# B&R Automation Studio project TD52 (part 22)

### module_AG.typ
```iecst
TYPE
	IN_AG_struct : 	STRUCT
		bCust_Dem_FreshOilPump : BOOL; (*Customized demand for fresh oil pump*) (*OldName:new V4.14; Cycle:5*)
		bCust_Dem_WasteOilPump : BOOL; (*Customized demand for waste oil pump*) (*OldName:new V4.14; Cycle:5*)
		bCust_Dem_OilFillValve : BOOL; (*Customized demand for oil fill valve*) (*OldName:new V4.14; Cycle:5*)
		bMsg1061 : BOOL; (* *) (*OldName:; Cycle:;*)
		tL_FreshOilTank : HALioAi_Type; (*Tank Level measurement input*) (*OldName: NewPv V4.12*)
		tL_WasteOilTank : HALioAi_Type; (*Tank Level measurement input*) (*OldName: NewPv V4.12*)
		tL_DayOilTank : HALioAi_Type; (*Tank Level measurement input*) (*OldName: NewPv V4.12*)
		tCDP_Op : HALioDi_Type; (*Di condensor pump failure*) (*OldName:GCB_ON; Cycle:5*)
		tFOP_Op : HALioDi_Type; (*DI fresh oil pump operating*) (*OldName:GCB_ON; Cycle:5*)
		tL_DayOilSump_Hi : HALioDi_Type; (*DI day oil tank oil collector pan high*) (*OldName:GCB_ON; Cycle:5*)
		tDayOilTank_Leck : HALioDi_Type; (*DI leckage day oil tank*) (*OldName:GCB_ON; Cycle:5*)
		tL_DayOilTank_Hi : HALioDi_Type; (*DI day oil tank high*) (*OldName:GCB_ON; Cycle:5*)
		tAuxV_Aux_ok : HALioDi_Type; (*DI voltage ok auxiliaries panel*) (*OldName:GCB_ON; Cycle:5*)
		tAuxV_ModIf_ok : HALioDi_Type; (*DI release auxiliaries module interface*) (*OldName:GCB_ON; Cycle:5*)
		tAB2AG : AmmBase2MM; (*AmmBase2MM*) (*OldName:new; Cycle:5*)
		tPB2MM : ParaBase2MM_type; (*ParaBase2MM*) (*OldName:new; Cycle:5*)
		iIdx_OMSS : INT; (*engine operation mode selection*) (*OldName:new; Cycle:5*)
		bIgn_Run : BOOL; (*ignition operating*) (*OldName:ZIB; Cycle:5*)
		bDemScavVa : BOOL; (* demand scavenging valve *) (*OldName:ANF_SPKL; Cycle:5*)
		b_ST_DemIgn : BOOL; (* Demand starter from ignition *) (*OldName:STARTER_IgnST; Cycle:5*)
		bBlocDelay_ManStart : BOOL; (* delay time next manual start *) (*OldName:T26; Cycle:5*)
		bECW_PreH_Dem_Customized : BOOL; (* engine cooling water preheating demand customized *) (*OldName:new; Cycle:5*)
		bEng_Aux_Dem_TOF : BOOL; (* demand auxiliaries with cool down time *) (*OldName:T12; Cycle:5*)
		bEG_BoVaOpened : BOOL; (* exhaust gas boiler valve opened *) (*OldName:M_KKAUF; Cycle:5*)
		bEG_ByVaOpened : BOOL; (* exhaust gas bypass valve opened *) (*OldName:M_BKAUF; Cycle:5*)
		bEO_PrelubeDemIgn : BOOL; (* demand Prelubricating from ignition *) (*OldName:PRELUBE_IgnST; Cycle:5*)
		tGCB_On : HALioDi_Type; (*DI generator circuit breaker closed*) (*OldName:GCB_ON; Cycle:5*)
		bGT_Rel : BOOL; (* Release gas train *) (*OldName:FG_GST; Cycle:5*)
		bGT_TypSwhActive : BOOL; (* Gas type switching active *) (*OldName:GASUM; Cycle:5*)
		bGT1_Check : BOOL; (* Gas train check 1 *) (*OldName:T88; Cycle:5*)
		bGT1_CheckOK : BOOL; (* Gas train 1 check OK *) (*OldName:M_GAS1OK; Cycle:5*)
		bGT2_Check : BOOL; (* Gas train check 2 *) (*OldName:T90; Cycle:5*)
		bGT2_CheckOK : BOOL; (* Gas train 2 check OK *) (*OldName:M_GAS2OK; Cycle:5*)
		bEng_Aux_Dem : BOOL; (*engine auxiliaries demand*) (*OldName:M_ANFHBT; Cycle:5*)
		bEng_Aux_Dem_CDR : BOOL; (*engine auxiliaries demand with cool down run*) (*OldName:ANFHBT; Cycle:5*)
		bEng_Dem : BOOL; (* module demanded *) (*OldName:M_AGFD; Cycle:5*)
		bEng_Dem_Aut_SUpF : BOOL; (* engine demand automatic startup failure *) (*OldName:BRI; Cycle:5*)
		bEng_Dem_Man_SUpF : BOOL; (* engine demand manual startup failure *) (*OldName:BRI_H; Cycle:5*)
		bEng_Dem_EPS : BOOL; (* engine demand for emergency operation *) (*OldName:M_NANF; Cycle:5*)
		bEng_Dem_Man : BOOL; (* engine demand manual *) (*OldName:M_ANF_H; Cycle:5*)
		bEng_MonOff : BOOL; (* engine monitoring OFF at startup *) (*OldName:T9; Cycle:5*)
		bEng_Rel : BOOL; (* engine release *) (*OldName:M_FG_MOT; Cycle:5*)
		bEng_RPSDem : BOOL; (* engine demanded  *) (*OldName:A_AGFD; Cycle:5*)
		tEng_Run : HALioDo_Type; (* engine operating state *) (*OldName:BTRB; Cycle:5*)
		bEng_SU_Man : BOOL; (* engine startup manual *) (*OldName:M_HSTART; Cycle:5*)
		bEng_SU_Aut : BOOL; (* engine startup automatic *) (*OldName:M7_6; Cycle:5*)
		bGV_On : BOOL; (* command open gas valves *) (*OldName:M_GASV; Cycle:5*)
		bMainsReturn : BOOL; (* mains return *) (*OldName:NWK; Cycle:5*)
		tMCB_On : HALioDi_Type; (*DI mains circuit breaker closed*) (*OldName:MCB_ON; Cycle:5*)
		bMsg1019 : BOOL; (* pressure engine cooling water low *) (*OldName:M_KDMI; Cycle:5*)
		bMsg1027 : BOOL; (* failure gas train 1 *) (*OldName:M_GST1; Cycle:5*)
		bMsg1029 : BOOL; (* failure gas train 2 *) (*OldName:M_GST2; Cycle:5*)
		bMsg1031 : BOOL; (* safety loop *) (*OldName:M_SIS; Cycle:5*)
		bN2_ScavCoPrelubeOn : BOOL; (* N2 scavenging command prelubrication ON *) (*OldName:PRELUBE_SC; Cycle:5*)
		bN2_ScavCoStarterOn : BOOL; (* N2 scavening command starter ON *) (*OldName:STARTER_SC; Cycle:5*)
		bOnly_Island : BOOL; (* only island operation *) (*OldName:REIN_INSEL; Cycle:5*)
		bOtherGenParallel : BOOL; (* other generator parallel *) (*OldName:other_gen_parallel; Cycle:5*)
		bP_Red_Active : BOOL; (* power reduction active - any kind *) (*OldName:PredAkt; Cycle:5*)
		bRel_ScavN2 : BOOL; (* conditions for scavenge with N2 *) (*OldName:FG_N2; Cycle:5*)
		bRelEngOp_OilSkid : BOOL; (*release engine operation from Oil Skid*) (*OldName:rel_EngOp_LOS; Cycle:5*)
		bRelEngTurn_OilSkid : BOOL; (*release engine barring gear (Durchdrehvorrichtung) from Oil Skid*) (*OldName:tPr_GenJOS_Ok; Cycle:5*)
		bScavFinished : BOOL; (* scavenging cycle finished  *) (*OldName:SPUEL_AB; Cycle:5*)
		tScavVaClosed : HALioDi_Type; (*DI scavenging valve closed*) (*OldName:SPK_ZU; Cycle:5*)
		rN_EngAct : REAL; (* engine speed actual [1/min] *) (*OldName:n_ist; Cycle:5*)
		rP_Act_Norm_Filt : REAL; (* actual power related to rP_Nom filtered T=1s *) (*OldName:P_IST; Cycle:5*)
		tAuxV_Eng_ok : HALioDi_Type; (* DI auxiliary voltage engine ok *) (*OldName:DI_AuxV_Eng_ok; Cycle:5*)
		tCCWP_Op : HALioDi_Type; (* DI charge cooling water pump operating (P.07-M-003) *) (*OldName:RM_GKP; Cycle:5*)
		tECWPrehV_Opened : HALioDi_Type; (* DI engine cooling water preheating valve opened *) (*OldName:new; Cycle:5*)
		tECWP_FC_Rdy : HALioDi_Type; (* DI engine cooling water pump frequency converter ready for operation *) (*OldName:MKP_FU_rdy; Cycle:5*)
		tECWP_Op : HALioDi_Type; (* DI engine cooling water pump operating *) (*OldName:RM_MKWP; Cycle:5*)
		tEngTurn : HALioDi_Type; (* DI engine turn equipment active *) (*OldName:DI_TURN1; Cycle:5*)
		tEngTurn2 : HALioDi_Type; (* DI engine turn equipment active *) (*OldName:DI_TURN2; Cycle:5*)
		tEO_Level_Hi : HALioDi_Type; (* DI engine oil level high from level switch  *) (*OldName:OMAX; Cycle:5*)
		tEO_Level_Lo : HALioDi_Type; (* DI engine oil level low from level switch  *) (*OldName:OMIN; Cycle:5*)
		tEO_Level_Lo_TC2 : HALioDi_Type; (* DI engine oil level low from level switch  *) (*OldName:OMIN; Cycle:2*)
		tEO_Refill : HALioDi_Type; (* DI engine oil refill ON from level switch *) (*OldName:OELV; Cycle:5*)
		tEOP_DemExt : HALioDi_Type; (* DI engine oil pump demand from external *) (*OldName:ANF_NKOP; Cycle:5*)
		tEOP_Op : HALioDi_Type; (* DI engine oil pump operating *) (*OldName:RM_VSP; Cycle:5*)
		tEOP1AC_CB_trip : HALioDi_Type; (* DI engine oil pump 1 AC circuit breaker trip *) (*OldName:DI_EOP1AC_CB_trip; Cycle:5*)
		tFireAlarm : HALioDi_Type; (* DI fire alarm *) (*OldName:BAL; Cycle:5*)
		tFS_ECW : HALioDi_Type; (* DI flow switch engine cooling water *) (*OldName:DI_FS_ECW; Cycle:5*)
		tGasAlarm : HALioDi_Type; (* DI gas alarm *) (*OldName:GAL; Cycle:5*)
		tGasPreAlarm : HALioDi_Type; (* DI gas pre alarm *) (*OldName:GALV; Cycle:5*)
		tGF_OilSystem : HALioDi_Type; (*DI general failure oil system*) (*OldName:newPV; Cycle:5*) (*STM 2*)
		tGT1_SafeDevOK : HALioDi_Type; (* DI Gassafety device 1 *) (*OldName:F_GAS1; Cycle:5*)
		tGT2_SafeDevOK : HALioDi_Type; (* DI Gassafety device 2 *) (*OldName:F_GAS2; Cycle:5*)
		tHWP_Op : HALioDi_Type; (* DI heating water pump operating (P.06-M-001) *) (*OldName:RM_HWP; Cycle:5*)
		tL_FreshOilTank_Hi : HALioDi_Type; (*DI fresh oil tank level high*) (*OldName:newPV; Cycle:5*) (*STM 2*)
		tLeak_FreshOilPump : HALioDi_Type; (*DI leakage fresh oil pump*) (*OldName:newPV; Cycle:5*) (*STM 2*)
		tLeak_FreshOilTank : HALioDi_Type; (*DI leakage fresh oil tank*) (*OldName:newPV; Cycle:5*) (*STM 2*)
		tLeak_WasteOilPump : HALioDi_Type; (*DI leakage waste oil pump*) (*OldName:newPV; Cycle:5*) (*STM 2*)
		tLeak_WasteOilTank : HALioDi_Type; (*DI leakage waste oil tank*) (*OldName:newPV; Cycle:5*) (*STM 2*)
		tMainsStartDevFail : HALioDi_Type; (* DI mains start device failure *) (*OldName:ST_NST; Cycle:5*)
		tMainsStartDevOk : HALioDi_Type; (* DI mains starting device OK *) (*OldName:FG_NST; Cycle:5*)
		tN2_GV1_Closed : HALioDi_Type; (* DI N2 gas valve 1 closed status *) (*OldName:N2V1_ZU; Cycle:5*)
		tN2_GV2_Closed : HALioDi_Type; (* DI N2 gas valve 2 closed status *) (*OldName:N2V2_ZU; Cycle:5*)
		tInAirER_Lou1Opened : HALioDi_Type; (* DI intake air engine room louver 1 opened*) (*OldName:ZJAL1_O; Cycle:5*)
		tInAirER_Lou2Opened : HALioDi_Type; (* DI intake air engine room louver 2 opened*) (*OldName:ZJAL2_O; Cycle:5*)
		tOF_FreshOilTank : HALioDi_Type; (*DI overfill prevention device fresh oil tank*) (*OldName:newPV; Cycle:5*) (*STM 2*)
		tOF_WasteOilTank : HALioDi_Type; (*DI overfill prevention device waste oil tank*) (*OldName:newPV; Cycle:5*) (*STM 2*)
		tOutAirER_LouOpened : HALioDi_Type; (* DI outlet air engine room louver opened*) (*OldName:AJAL_O; Cycle:5*)
		tP_Heat_Imp : HALioDi_Type; (*heating power engine heat water circuit impulse*) (*STM 2*)
		tPr_CC : HALioAi_Type; (* AI pressure crank case [bar] *) (*OldName:AI_KGD; Cycle:5*)
		tPr_EngLubOil : HALioAi_Type; (*AI: Oil pressure engine lube oil - last lubr. point [bar] M.03-PI-001*) (*OldName:ODR_WE; Cycle:5*)
		tRelAux : HALioDi_Type; (* DI release engine operation from auxiliaries with monitoring *) (*OldName:FG_HBT; Cycle:5*)
		tRelAuxNoMon : HALioDi_Type; (* DI release engine operation from auxiliaries without bridging for blackout start *) (*OldName:FG_HBT2; Cycle:5*)
		tRelMainGVext : HALioDi_Type; (* DI release main gas valve from external *) (*OldName:FG_HGV_ext; Cycle:5*)
		tT_ECW : HALioAi_Type; (* AI temperature engine cooling water [°C] M.04-TI-001 *) (*OldName:ANA.KWT; Cycle:5*)
		tT_ECW_Mod_In : HALioAi_Type; (*temperature engine cooling water, engine cooling water module inlet M.04-TI-003*) (*OldName:newPv; Cycle:5;*)
		tT_ECW_PreH_Hi : HALioDi_Type; (* TS: temperature engine cooling water preheating high M.04-TI-081*) (*OldName:mkw_preh_warn; Cycle:5*)
		tT_ECW_PreH_HiHi : HALioDi_Type; (* TS: temperature engine cooling water preheating high high M.04-TI-026*) (*OldName:mkw_preh_alarm; Cycle:5*)
		tTCOP_Op : HALioDi_Type; (* DI turbo charger oil pump operating *) (*OldName:RM_TLP; Cycle:5*)
		tU_StarterBat_Lo : HALioDi_Type; (* DI voltage starter battery low *) (*OldName:STBM; Cycle:5*)
		tU_Starter_engage1 : HALioAi_Type; (*Start motor 1 function voltage*)
		tU_Starter_engage2 : HALioAi_Type; (*Start motor 2 function voltage*)
		tU_Starter_engage3 : HALioAi_Type; (*Start motor 3 function voltage*)
		tAuxFail : HALioDi_Type; (*DI auxilaries failure*) (*OldName:ST_HBT; Cycle:5*)
		tECW_PreHV_Closed : HALioDi_Type; (*DI engine cooling water preheating valve status closed M.04-YCS-002*) (*OldName:DI_ECWV_Closed; Cycle:5*)
		tECW_PreHV_Opened : HALioDi_Type; (*DI engine cooling water preheating valve status opened M.04-YCS-002*) (*OldName:DI_ECWV_Open; Cycle:5*)
		tL_ECW_Lo : HALioDi_Type; (*DI engine cooling water level low*) (*OldName:KSMI_W; Cycle:5*)
		tL_ECW_LoLo : HALioDi_Type; (*DI engine cooling water level low low*) (*OldName:KSMI; Cycle:5*)
		tEngStartFailure : HALioDi_Type; (*DI engine start failure*) (*OldName:ANLST; Cycle:5*)
		tTransformerWarning : HALioDi_Type; (*DI transformer failure*) (*OldName:ST_TR_W; Cycle:5*)
		tTransformerTrip : HALioDi_Type; (*DI transformer failure*) (*OldName:ST_TR; Cycle:5*)
		tCP_CBTrip : HALioDi_Type; (*DI module and/or interface control panel - circuit breaker tripped*) (*OldName:SIFA_IA; Cycle:5*)
		tIFCP_CBTrip : HALioDi_Type; (*DI interface control panel - circuit breaker tripped*) (*OldName:SIFA_I; Cycle:5*)
		tMCP_CBTrip : HALioDi_Type; (*DI module control panel - circuit breaker tripped*) (*OldName:SIFA_A; Cycle:5*)
		tSafetyLoop_Gas : HALioDi_Type; (*DI safety loop gas ok*) (*OldName:DI_Gas_SL; Cycle:5*)
		tGV1_Open : HALioDo_Type; (*DO open gas valve 1*) (*OldName:GASV1; Cycle:5*)
		tGV2_Open : HALioDo_Type; (*SAFETY PLC: DO open gas valve 2*) (*OldName:GASV2; Cycle:5*) (*V04.14.00.00*)
		tGV3_Open : HALioDo_Type; (*SAFETY PLC: DO open gas valve 3*) (*OldName: new PV; Cycle: 5;*) (*V04.25.00.00*)
		tGV4_Open : HALioDo_Type; (*SAFETY PLC: DO open gas valve 4*) (*OldName: new PV; Cycle: 5;*) (*V04.25.00.00*)
		tDCGA_GV_Open : HALioDo_Type; (*SAFETY PLC: DO open gas valve for decentral gas addition*) (*OldName: new PV; Cycle: 5;*) (*V04.25.00.00*)
		tL_FreshOilTank_Lo : HALioDi_Type; (*DI fresh oil tank level low*) (*OldName:FOTMI; Cycle:5*)
		tL_WasteOilTank_Hi : HALioDi_Type; (*DI waste oil tank level high*) (*OldName:AOTMA; Cycle:5*)
		tAuxOverVoltProt_Ok : HALioDi_Type; (*failure over voltage protection auxiliaries power supply*) (*OldName:DI_AOVP; Cycle:5*)
		tUPS_Ok : HALioDi_Type; (*uninterrupted power supply ok/alarm*) (*OldName:DI_USV_OK; Cycle:5*)
		tSafetyLoop_Eng : HALioDi_Type; (*safety loop engine ok*) (*OldName:RUHE; Cycle:5*)
		tSafetyLoop_EmStop : HALioDi_Type; (*safety loop emergency stop ok*) (*OldName:DI_SIS; Cycle:5*)
		tSafetyLoop_HWC : HALioDi_Type; (*safety loop heat water circuit ok*) (*OldName:RM_HK; Cycle:5*)
		tPr_HW_Lo : HALioDi_Type; (*DI heat water pressure low*) (*OldName:HWD; Cycle:5*)
		tPr_HW_Hi1 : HALioDi_Type; (*DI heat water pressure high*) (*OldName:HWDX1; Cycle:5*)
		tPr_HW_Hi : HALioDi_Type; (*DI heat water pressure high*) (*OldName:HWDX; Cycle:5*)
		tT_HW_Hi1 : HALioDi_Type; (*DI heat water temperature high*) (*OldName:HWTP1; Cycle:5*)
		tT_HW_Hi : HALioDi_Type; (*DI heat water temperature high*) (*OldName:HWTP; Cycle:5*)
		tT_AirIFCP_Hi : HALioDi_Type; (*DI air temperature interface control panel high*) (*OldName:MCP_TEMP; Cycle:5*)
		tPr_TC_EOF_After : HALioAi_Type; (*AI oil pressure after turbocharger oil filter, J920: NUP62/M.03-PI-062 // J6: M.03-PI-063*) (*OldName:OilPress_a_ATL_f; Cycle:5*)
		tEOF_DiffMax : HALioDi_Type; (*DI: Oil filter differential pressure maximum E.03-PDS-001*) (*OldName:ODFM; Cycle:5*)
		tPr_TCOF_EOF_DiffMax : HALioDi_Type; (*DI: Turbo charger oil filter differential pressure maximum M.03-PDS-001*) (*OldName:DI_dp_TCOF_hi; Cycle:5*)
		tPr_EO_Gear_Min : HALioDi_Type; (*DI: Oil pressure low transmission*) (*OldName:GO_DMI; Cycle:5*)
		tT_EO_Gear_Max : HALioDi_Type; (*DI: Oil temperature high transmission*) (*OldName:GO_TMA; Cycle:5*)
		tEO_Supply_Fail : HALioDi_Type; (*DI: Oil supply failure*) (*OldName:ST_OELV; Cycle:5*)
		tPr_EOF_DiffMon : HALioAi_Type; (*AI: Oil pressure before oil filter [bar] M.03-PI-002 (NUP29)*) (*OldName:ssOilPbFilter; OilPress_f_f; Cycle:5*)
		tPr_EOF_After : HALioAi_Type; (*AI: Oil pressure after oil filter [bar] M.03-PI-057 (NUP57)*) (*OldName:OilPress_a_f; Cycle:5*)
		tEO_Quality : HALioAi_Type; (*AI: Oil quality sensor, QTOil1/ AI_ *) (*OldName:OilQual; Cycle:5*)
		tPr_TC_EOF_Before : HALioAi_Type; (*AI: Oil pressure in front of turbocharger oil filter, NUP61/M.03-PI-061*) (*OldName:OilPress_f_ATL_f; Cycle:5*)
		tEO_Level : HALioAi_Type; (*AI: Oil fill level, LS5/M.03-LI-001*) (*OldName:Oil_Fill; Cycle:5*)
		tT_EO : HALioAi_Type; (*AI: Oil temperature M.03-TI-001*) (*OldName:ANA.OTP; Cycle:5*)
		tT_EO_Mod_Out : HALioAi_Type; (*temperature engine oil, oil module outlet M.03-TI-003*) (*OldName:newPv; Cycle:5;*)
		tCnt_Oil_NC150 : HALioAi_Type; (*AI oil counter*) (*OldName:AIOilCounter; Cycle:2*)
		tCnt_Oil_DC2395 : HALioAi_INT_Type; (*AI oil counter circular buffer*) (*OldName:AIOilCounterCircle; Cycle:2*)
		iCnt_OpHours : DINT; (*Operating hours *) (*OldName:betrieb_h; Cycle:5*)
		rP_Nom : REAL; (*Nominal electric power [kW], depends on gastype*) (*OldName:p_nenn; Cycle:5*)
		tT_EO_Preheating : HALioAi_Type; (*engine oil temperature preheating, NUT78/M.03-TI-078*) (*OldName:OilTemp_preh; Cycle:5*)
		tT_EO_Pan : HALioAi_Type; (*engine oil temperature oil pan, M.03-TI-002*) (*OldName:AI_t_OilPan; Cycle:5*)
		tT_EO_PreH_Hi : HALioDi_Type; (*engine oil preheating max.warning(temp.limiter) M.03-TS-072*) (*OldName:DI_EO_PreH_w; Cycle:5*)
		tT_EO_PreH_HiHi : HALioDi_Type; (*engine oil preheating max.alarm(temp.limiter) M.03-TS-080*) (*OldName:DI_EO_PreH_a; Cycle:5*)
		tT_EOP_After : HALioAi_Type; (*engine oil temperature after  oil pump, NUT71/M.03-TI-071*) (*OldName:AI_t_EOaPump; Cycle:5*)
		tCnt_OilPulse : HALioDi_Type; (*DI oil counter*) (*OldName:DI_OilCount; Cycle:2*)
		bMsg3003 : BOOL; (*Common measuring signal failure A3003*) (*OldName:M_MS ; Cycle:5*)
		tEOP_FC_Rdy : HALioDi_Type; (*DI: engine oil pump freq.converter operation/ready*) (*OldName:VSP_FU_rdy; Cycle:5*)
		bMsg3361 : BOOL; (*failure gas train 1 - line 4*) (*OldName:M_GST1_4; Cycle:5;*)
		bMsg3360 : BOOL; (*failure gas train 1 - line 3*) (*OldName:M_GST1_3; Cycle:5;*)
		bMsg3359 : BOOL; (*failure gas train 1 - line 2*) (*OldName:M_GST1_2; Cycle:5;*)
		tL_OilSumpHi : HALioDi_Type; (*DI level oil sump high*) (*OldName:DI_LS_OilSumpHi; Cycle:5;*)
		tL_OilSump2Hi : HALioDi_Type; (*DI level oil sump 2 high*) (*OldName:DI_LS_OilSump2Hi; Cycle:5;*)
		tL_OilSump3Hi : HALioDi_Type; (*DI level oil sump 3 high*) (*OldName:newpv; Cycle:5;*)
		tCO_Alarm : HALioDi_Type; (*DI CO alarm*) (*OldName:DI_CO_alarm; Cycle:5;*)
		tCO_PreAlarm : HALioDi_Type; (*DI CO prealarm*) (*OldName:DI_CO_prealarm; Cycle:5;*)
		tAuxErrWarn : HALioDi_Type; (*DI auxiliaries error*) (*OldName:DI_HBTW; Cycle:5;*)
		tActFiltAlarm : HALioDi_Type; (*DI activ filter alarm*) (*OldName:DI_FIL_A; Cycle:5;*)
		tActFiltWarn : HALioDi_Type; (*DI activ filter warning*) (*OldName:DI_FIL_W; Cycle:5;*)
		tL_InMa_NotHi : HALioDi_Type; (*DI water ingress into inlet manifold negated*) (*OldName:DI_LS2ChC; Cycle:5;*)
		tL_InMa_Hi : HALioDi_Type; (*DI water ingress into inlet manifold*) (*OldName:DI_LS4ChC; Cycle:5;*)
		tImp_OpHour : HALioDo_Type; (*DO: Impulse for operation hour counter *) (*OldName:M_BTRIMP,H_IMP;Cycle:5;*)
		iCnt_Starts : DINT; (* = STRT_high - IF543 start counter*) (*OldName:C; Cycle:5;*)
		iPassLevel : INT; (*pass level actual*) (*OldName:ucPassLevel; Cycle:5;*)
		bGrC_HBErr_AUS : BOOL := FALSE; (*TRUE = Störung HB A1129 deaktiviert über GCEvent*) (*OldName:bGC_HBErr_AUS;*)
		rCust_SparePara : ARRAY[0..200]OF REAL; (*SPS_REZP1 to SPS_REZP200*) (*OldName:SPS_REZP1, SPS_REZP2, SPS_REZP70; Cycle: 5;*)
		tCustAnaIn : ARRAY[0..120]OF HALioAi_Type; (*Replacement for RAN_KANAL...*) (*OldName:ANA_RAN; Cycle: 5;*)
		tCustDigIn : ARRAY[0..200]OF HALioDi_Type; (*new, reserved for Project specific use*) (*OldName:new PV; Cycle: 5;*)
		bEng_Bloc_SGM : BOOL; (*SGM blocks engine start because reference procedure is active*) (*OldName:M_GM_Ref; Cyclic:5;*)
		bGT1_SafeDevOK : BOOL; (*Gassafety device 1 release (From DI and task)*) (* OldName:F_GAS1; Cyclic:5;*)
		tTCOP_Grid : HALioDi_Type; (*TC oil pump power supply ok*) (*OldName:DI_TCOP_NETZ; Cycle:5;*)
		tPr_Oil_LPTC_In_A : HALioAi_Type; (*oil pressure LP turbo charger A inlet M.03-PI-101*) (*OldName:P_OEL_ND_EintrittA; Cycle:5;*)
		tPr_Oil_LPTC_In_B : HALioAi_Type; (*oil pressure LP turbo charger B inlet M.03-PI-201*) (*OldName:P_OEL_ND_EintrittB; Cycle:5;*)
		tBbBlower_FC_Rdy : HALioDi_Type; (*DI Blow-by Blower FC ready *) (* Oldname:new PV , Cycle:5 *)
		tPr_f_BbFilt : HALioAi_Type; (*AI Pressure before Blow-by filter M.03-PI-003*) (* Oldname: newPV, Cycle:5 *)
		tPr_f_BbFilt_A : HALioAi_Type; (*AI Pressure before Blow-by filter M.03-PI-103*) (* Oldname: newPV, Cycle:5 *)
		tPr_f_BbFilt_B : HALioAi_Type; (*AI Pressure before Blow-by filter M.03-PI-203*) (* Oldname: newPV, Cycle:5 *)
		tPr_a_BbFilt : HALioAi_Type; (*AI Pressure after Blow-by filter M.03-PI-004*) (* Oldname:newPV , Cycle:5 *)
		tPr_a_BbFilt_A : HALioAi_Type; (*AI Pressure after Blow-by filter M.03-PI-104*) (* Oldname:newPV , Cycle:5 *)
		tPr_a_BbFilt_B : HALioAi_Type; (*AI Pressure after Blow-by filter M.03-PI-204*) (* Oldname:newPV , Cycle:5 *)
		tCV_Eng_Low : HALioDi_Type; (*control voltage low - engine*) (*OldName:DI_CV_ENG_low; Cycle:5;*)
		tCV_TCA_Low : HALioDi_Type; (*control voltage low - turbo charger aux.*) (*OldName:DI_CV_TCA_low; Cycle:5;*)
		tCV_MCP_Low : HALioDi_Type; (*control voltage low - module control panel*) (*OldName:DI_CV_MCP_low; Cycle:5;*)
		tPr_AirStarter_Tank : HALioAi_Type; (*AI air starter tank pressure [bar] (P.31-PI-001)*) (* Oldname:new PV , Cycle:5 *)
		tTCOP_CB_On : HALioDi_Type; (*prelubrication pump turbo charger circuit breaker on*) (*OldName:DI_TCOP_CB_trip; Cycle:5;*)
		tPr_AirStarter_Supply : HALioAi_Type; (*Air starter supply pressure [bar] (E.31-PI-001)*) (* Oldname:new PV , Cycle:5 *)
		tCnt_N_AirStarter : HALioAi_INT_Type; (*AI - counter modul- air starter speed [rpm] (E.00-SI-006)*) (* Oldname:new PV , Cycle:5 *)
		tTCOP_UPS_CB_On : HALioDi_Type; (*prelubrication pump turbo charger USV circuit breaker on*) (*OldName:DI_TCOP_USV_OK; Cycle:5;*)
		tECWP_PreH_CB_On : HALioDi_Type; (*preheating pump circuit breaker on*) (*OldName:DI_ECWP_PreH_CB_trip; Cycle:5;*)
		tChUnit1_CB_On : HALioDi_Type; (*charging unit turbo charger auxiliaries circuit breaker on*) (*OldName:DI_LG1_CB_trip; Cycle:5;*)
		tChUnit2_CB_On : HALioDi_Type; (*charging unit turbo charger auxiliaries circuit breaker on*) (*OldName:DI_LG2_CB_trip; Cycle:5;*)
		tChUnit3_CB_On : HALioDi_Type; (*charging unit engine interface panel circuit breaker on*) (*OldName:DI_LG3_CB_trip; Cycle:5;*)
		tChUnit4_CB_On : HALioDi_Type; (*charging unit engine interface panel circuit breaker on*) (*OldName:DI_LG4_CB_trip; Cycle:5;*)
		tENGIA_CB_On : HALioDi_Type; (*power supply engine interface panel circuit breaker on*) (*OldName:DI_ENGIA_CB_trip; Cycle:5;*)
		tECWP_Service_CB_On : HALioDi_Type; (*service cooling water pump circuit breaker on*) (*OldName:DI_ECWP_ServCB_trip; Cycle:5;*)
		tPS400V_ENGIA_CB_On : HALioDi_Type; (*engine interface panel AC power supply circuit breaker on*) (*OldName:DI_HS400V_ENGIA; Cycle:5;*)
		tUPS_CB_On : HALioDi_Type; (*UPS circuit breaker  on*) (*OldName:DI_USV_CB_trip; Cycle:5;*)
		tENGIA_UPS_CB_On : HALioDi_Type; (*engine interface panel UPS supply circuit breaker on*) (*OldName:DI_ENGIA_USV_CB_trip; Cycle:5;*)
		tECWP_Service_COn : HALioDi_Type; (*engine cooling water service pump command ON*) (*OldName:DI_ECWP_ServMOC; Cycle:5;*)
		tECWV_Fail : HALioDi_Type; (*engine cooling water preheating valve failure*) (*OldName:DI_ECWV_FAIL; Cycle:5;*)
		tPS_EI_CB_On : HALioDi_Type; (*power supply engine interface panel circuit breaker on*) (*OldName:PS_EI_CB_trip; Cycle:5;*)
		tSTT_CB_On : HALioDi_Type; (*control voltage transformer circuit breaker on*) (*OldName:STT_CB_trip; Cycle:5;*)
		bMsg1056 : BOOL; (*safety loop - engine*) (*OldName:M_RUHE;Cycle:5;*)
		bMsg3404 : BOOL; (*water pressure cooler circuit low*) (*OldName:M_NKWD_W; Cycle:5;*)
		bMsg1130 : BOOL; (*charge cooler water pressure low*) (*OldName:AMM_A11xx[]; Cycle:5;*)
		bMsg2117 : BOOL; (*charge cooler water pressure low*) (*OldName:M_GKWD; Cycle:5;*)
		tEG_ByVaOpened : HALioDi_Type; (*DI exhaust gas bypass valve opened*) (*OldName:BK_AUF;Cycle:5*)
		tEG_ByVaClosed : HALioDi_Type; (*DI exhaust gas bypass valve closed*) (*OldName:BK_ZU;Cycle:5*)
		tEG_BoVaOpened : HALioDi_Type; (*DI exhaust gas boiler valve opened*) (*OldName:KK_AUF;Cycle:5*)
		tEG_BoVaClosed : HALioDi_Type; (*DI exhaust gas boiler valve closed*) (*OldName:KK_ZU;Cycle:5*)
		tCV_GENI_Ok : HALioDi_Type; (*control voltage missing generator interface*) (*OldName:DI_CV_GENI_ok;Cycle:5*)
		tCV_ENGIB_Ok : HALioDi_Type; (*control voltage missing engine interface bank B*) (*OldName:DI_CV_ENGIB_ok;Cycle:5*)
		tCV_TCMI_Ok : HALioDi_Type; (*control voltage missing turbo charger module interface *) (*OldName:DI_CV_TCMI_ok;Cycle:5*)
		tCV_TCUS_Ok : HALioDi_Type; (*control voltage missing turbo charger unit sensor cabinet *) (*OldName:DI_CV_TCUS_ok;Cycle:5*)
		tCV_JWMI_Ok : HALioDi_Type; (*control voltage missing jacket water module interface *) (*OldName:DI_CV_JWMI_ok;Cycle:5*)
		tCV_OILMI_Ok : HALioDi_Type; (*control voltage missing oil module interface *) (*OldName:DI_CV_OILMI_ok;Cycle:5*)
		tCV_M_Ok : HALioDi_Type; (*control voltage missing module interface cabinet*) (*OldName:DI_CV_M_ok;Cycle:5*)
		tCV_A_Ok : HALioDi_Type; (*control voltage missing module control cabinet *) (*OldName:DI_CV_A_ok;Cycle:5*)
		tCV_AUX_Ok : ARRAY[0..5]OF HALioDi_Type; (*control voltage missing auxiliaries control cabinet*) (*OldName:DI_CV_AUX_ok;Cycle:5*)
		tPr_EOaP : HALioAi_Type; (*engine oil pressure after pump M.03-PI-007*) (*Oldname:newPV;Cycle:5*)
		tPS_EOaP_HiHi : HALioDi_Type; (*engine oil pressure after pump high safety pressure switch M.03-PS-001*) (*Oldname:newPV;Cycle:5*)
		tPr_OFUbFilt : HALioAi_Type; (*pressure oil filter unit before filter M.03-PI-011*) (*Oldname:newPV;Cycle:5*)
		tPr_OFUaFilt : HALioAi_Type; (*pressure oil filter unit after filter M.03-PI-012*) (*Oldname:newPV;Cycle:5*)
		bGridCode_ON : BOOL; (*any dyn. GridCode function activated*)
		bServiceMode : BOOL; (*service mode*) (*OldName:bServiceBegin; Cycle:5;*)
		bImp_Start : BOOL; (*impulse for start counter*) (*OldName:T25,M_STRTIMP;Cycle:5;*)
		tPr_OFUbCentrifuge : HALioAi_Type; (*pressure oil filter unit before centrifuge M.03-PI-008*) (*Oldname:newPV;Cycle:5*)
		tOFUP_Filter_CB : HALioDi_Type; (*oil filter unit pump filter M.03-P-007 - circuit breaker*) (*Oldname:newPV;Cycle:5*)
		tOFUP_Centrifuge_CB : HALioDi_Type; (*oil filter unit pump centrifuge M.03-P-006 - circuit breaker*) (*Oldname:newPV;Cycle:5*)
		bSimWinMOD_Active : BOOL; (*WinMode simulation active *) (*OldName:new PV; Cycle:5*)
		bStop : BOOL; (*Manual op.mode engine stop button*) (*OldName:new PV; Cycle:5*)
		bStart : BOOL; (*Manual op.mode engine start button*) (*OldName:new PV; Cycle:5*)
		Pos_OutlLou2_OK : BOOL; (*position feedback air outlet louver 2 OK depending on parameter*)
		Pos_OutlLou1_OK : BOOL; (*position feedback air outlet louver 1 OK depending on parameter*)
		Pos_InlLou2_OK : BOOL; (*position feedback air inlet louver 2 OK depending on parameter*)
		Pos_InlLou1_OK : BOOL; (*position feedback air inlet louver 1 OK depending on parameter*)
		bPermPreLube_Dem : BOOL; (*Demand permanent prelubification to AuxiliariesGeneral*) (*OldName:new PV; Cycle:5*)
		tPr_TCO : HALioAi_Type; (*pressure oil before turbo charger M.03-PI-063*)
		tFastStartReq : HALioDi_Type; (*Fast Start Required*) (*OldName:newPV; Cycle:5;*)
		bFS_Act : BOOL; (*FastStart activated (enabled and required from customer)*) (*Oldname: new PV, Cycle:5*)
		tU_StarterBat : HALioAi_Type; (*AI starter battery voltage monitoring*)
		tEOP_BWS : HALioDi_Type; (*DI pre-lubrication engine oil pump brush wear signal*)
		tEOP_BWS2 : HALioDi_Type; (*DI pre-lubrication engine oil pump brush wear signal 2*)
		rCustomizedAG : ARRAY[0..99]OF REAL; (*New customizable interface 2017  - BETA PHASE, use only in coordination with TPSS*)
		rP_Act_Norm_Filt_TC2 : REAL; (*actual power related to rP_Nom filtered T=1s *) (*OldName:P_IST; Cycle:2*)
		tInAirER_Lou1Closed : HALioDi_Type; (*DI intake air engine room louver 1 Closed*)
		tInAirER_Lou2Closed : HALioDi_Type; (*DI intake air engine room louver 2 Closed*)
		tOutAirER_LouClosed : HALioDi_Type; (*DI outlet air engine room louver Closed*)
		bMsg9226 : BOOL; (*charge cooler 2 water pressure low*) (*OldName:newPV; Cycle:5;*)
		bMsg2684 : BOOL; (*Temperature heat water supply hydraulic engine cooling water preheating signal failure*) (*OldName:newPV; Cycle:5;*)
		tT_HW_Su_PreH_ECW : HALioAi_Type; (*AI Temperature hydraulic ECW pre-heating supply (J3+J4: P.06-TI-050, J920: M.04-TI-005)*) (*OldName:newPV; Cycle:5;*)
		tCC2WP_Op : HALioDi_Type; (*DI charge cooler 2 water pump operating (P.07-M-007)*) (*OldName:newPV; Cycle:5*)
		tHWP1_Op : HALioDi_Type; (*DI Redundant heating water pump 1 operating (P.06-M-001)*)
		tHWP2_Op : HALioDi_Type; (*DI Redundant heating water pump 2 operating (P.06-M-002)*)
		bCCWP_Dem : BOOL; (*Charge cooler water pump demand*)
		tCCWP1_Op : HALioDi_Type; (*DI Redundant charge cooler water pump 1 operating (P.07-M-003)*)
		tCCWP2_Op : HALioDi_Type; (*DI Redundant charge cooler water pump 2 operating (P.07-M-013)*)
		bCC2WP_Dem : BOOL; (*Charge cooler 2 water pump demand*)
		tCC2WP1_Op : HALioDi_Type; (*DI Redundant charge cooler 2 water pump 1 operating (P.07-M-007)*)
		tCC2WP2_Op : HALioDi_Type; (*DI Redundant charge cooler 2 water pump 2 operating (P.07-M-017)*)
		bEmCWP_Dem : BOOL; (*Emergency cooler water pump demand*)
		tEmCWP_Op : HALioDi_Type; (*DI Emergency cooler water pump operating (P.09-M-001)*)
		tEmCWP1_Op : HALioDi_Type; (*DI Redundant emergency cooler water pump 1 operating (P.09-M-001)*)
		tEmCWP2_Op : HALioDi_Type; (*DI Redundant emergency cooler water pump 2 operating (P.09-M-002)*)
		tBoilerFailure : HALioDi_Type; (*DI Boiler failure*)
		tSeismicAlarm : HALioDi_Type; (*DI Seismic alarm (M.00-AI-100)*)
		tFireProtFlap1_InlAir_Opened : HALioDi_Type; (*fireprotectionflap 1 inlet-air opened*)
		tFireProtFlap2_InlAir_Opened : HALioDi_Type; (*fireprotectionflap 2 inlet-air opened*)
		tFireProtFlap1_OutlAir_Opened : HALioDi_Type; (*fireprotectionflap 1 outlet-air opened*)
		tFireProtFlap2_OutlAir_Opened : HALioDi_Type; (*fireprotectionflap 2 outlet-air opened*)
		tFireProtFlap1_InlAir_Closed : HALioDi_Type; (*fireprotectionflap 1 inlet-air closed*)
		tFireProtFlap2_InlAir_Closed : HALioDi_Type; (*fireprotectionflap 2 inlet-air closed*)
		tFireProtFlap1_OutlAir_Closed : HALioDi_Type; (*fireprotectionflap 1 outlet-air closed*)
		tFireProtFlap2_OutlAir_Closed : HALioDi_Type; (*fireprotectionflap 2 outlet-air closed*)
		tPr_AirST_Engage : HALioAi_Type; (*AI Pressure air starter engagement [bar] (E.31-PI-004)*)
		bEng_Bloc : BOOL; (*Collective signal for engine start blockade*)
		tPr_ECW : HALioAi_Type; (*AI Engine cooling water pressure (M.04-PI-001)*)
		tPr_ECWaP1 : HALioAi_Type; (*AI Engine cooling water pressure after ECW pump 1 (M.04-PI-010)*)
		tPr_ECWaP2 : HALioAi_Type; (*AI Engine cooling water pressure after ECW pump 2 (M.04-PI-011)*)
		tECWP_CB_On : HALioDi_Type; (*DI Engine cooling water pump circuit breaker on*)
		tL_FreshOilTank_LoLo : HALioDi_Type; (*DI Fresh oil tank level low (2nd level switch)*)
		tL_DayOilTank_Lo : HALioDi_Type; (*DI Fresh oil day tank level low*)
		tL_DayOilTank_LoLo : HALioDi_Type; (*DI Fresh oil day tank level low (2nd level switch)*)
		tOF_DayOilTank : HALioDi_Type; (*DI Overfill prevention device fresh oil day tank*)
		tL_WasteOilDayTank_Hi : HALioDi_Type; (*DI Waste oil day tank level high*)
		tOF_WasteOilDayTank : HALioDi_Type; (*DI Overfill prevention device waste oil day tank*)
		tPS_FreshOilPump_Hi : HALioDi_Type; (*DI Fresh oil pump oil pressure maximum*)
		tT_HW_EGHE_Hi : HALioDi_Type; (*DI Heating water temperature max. exhaust gas cooler*)
		tT_HW_EGCD_Hi : HALioDi_Type; (*DI Heating water temperature max. exhaust gas condenser*)
		tCust_HW_Ext_Trip : HALioDi_Type; (*DI External heating water circuit monitoring*)
		tMCP_AuxPS_CB_Trip : HALioDi_Type; (*auxiliaries power supply circuit breaker module control panel tripped*)
		tMCP_AuxPS_CB_On : HALioDi_Type; (*auxiliaries power supply circuit breaker module control panel opened*)
		tMCP_AuxPS_GndFault : HALioDi_Type; (*earth fault auxiliaries power supply module control panel*)
		tMCP_FC_GndFault : HALioDi_Type; (*earth fault frequency converter module control panel*)
		tMIP_FC_GndFault : HALioDi_Type; (*earth fault frequency converter module interface panel*)
		tAuxCP_FC_GndFault : HALioDi_Type; (*earth fault frequency converter auxiliaries control panel*)
		tAuxCP_AuxPS_GndFault : HALioDi_Type; (*earth fault auxiliaries power supply auxiliaries control panel*)
		tAuxCP_AuxPS_CB_Trip : HALioDi_Type; (*auxiliaries power supply circuit breaker auxiliaries control panel tripped*)
		tAuxCP_AuxPS_CB_On : HALioDi_Type; (*auxiliaries power supply circuit breaker auxiliaries control panel opened*)
		rP_Set_Norm : REAL; (* power setpoint related to rP_Nom *) (*OldName:p_soll;Cycle:5;*)
		tU_BufferBat1 : HALioAi_Type; (*AI Buffer battery 1 voltage*)
		tU_BufferBat2 : HALioAi_Type; (*AI Buffer battery 2 voltage*)
		tBatChargeDev_Ok : HALioDi_Type; (*DI Status battery charging devices*)
		tLeak_OilExtensionTank1 : HALioDi_Type; (*DI Oil leakage detection additional oil tank 1 (P.03-LS-021)*)
		tLeak_OilExtensionTank2 : HALioDi_Type; (*DI Oil leakage detection additional oil tank 2 (P.03-LS-031)*)
		tLeak_OilExtensionTank3 : HALioDi_Type; (*DI Oil leakage detection additional oil tank 3 (P.03-LS-041)*)
		tU_CtrlBat : ARRAY[1..iNum_CtrlBatMon]OF HALioAi_Type; (*AI Control battery extension voltage*)
		tCtrlBat_ChargeDev_Ok : ARRAY[1..iNum_CtrlBatMon]OF HALioDi_Type; (*DI Status battery charging devices*)
		sLocIdent_CtrlBatMon : ARRAY[1..iNum_CtrlBatMon]OF STRING[10]; (*Control battery test set location*)
		bAuxV_ok_CtrlBatMon : ARRAY[1..iNum_CtrlBatMon]OF BOOL; (*Control battery test set status AuxV supply*)
		iCAN_OQS_OC_us_ident : UDINT; (*User ident for OQS OC sensor CAN interface*) (* OldName:new PV; Cycle:2*)
		bMsg1050 : BOOL; (*engine cooling water pressure high*) (*OldName:new PV; Cycle:5;*)
		bLR_ActSat_CBV : BOOL; (* load rejection flag for muting crankcase pressure max trip *) (*OldName:new PV; Cycle:5;*)
		tMnsOk : HALioDi_Type; (*DImainsok*)
		bMsg2101 : BOOL; (*signal failure engine cooling water temperature*) (*OldName:M_MSKWT; Cycle:5;*) (*V04.13.00.00*)
		bIgn_Run_CAN : BOOL; (*Ignition system is running - feedback from CAN*) (*V04.13.00.00*)
		bTOF_HwBypassDigitalTwin : BOOL; (*Hardware bypass digital twin - T3 adaptive cranking time*)
		bEng_Dem_Aut : BOOL; (*demand automatic mode *)
		bInLouRelVE : BOOL; (*inlet louvers open or not closed*)
		bSafetyPLC_Active : BOOL; (*SAFETY PLC: SafetyPLC is active*) (*OldName: new PV; Cycle: 5;*) (*V04.14.00.00*)
		rVol_PurgeAir_SafeOUT : REAL; (*SAFETY PLC: Volume of purge air*) (*OldName: new PV; Cycle: 5;*) (*V04.25.00.00*)
		bSafeOUT_Purge_OK : BOOL; (*SAFETY PLC: Purge state (true: engine purged, false: engine not purged)*) (*OldName: new PV; Cycle: 5;*) (*V04.25.00.00*)
		tGasSysErr : HALioDi_Type; (*DI System failure - Gas detection system (P.17-JI-200)*) (*OldName: new PV; Cycle: 5;*) (*V04.25.00.00*)
		tFireSysErr : HALioDi_Type; (*DI System failure - Fire detection system (P.17-JI-001)*) (*OldName: new PV; Cycle: 5;*) (*V04.25.00.00*)
		bRel_HWP_Dem : BOOL; (*SAFETY PLC: Release heating water pump*) (*OldName: new PV; Cycle: 5;*) (*V04.25.00.00*)
		bSafeOUT_GT1_SafeDevOK : BOOL; (*SAFETY PLC: Gas safety device 1 OK*) (*OldName: new PV; Cycle: 5;*) (*V04.25.00.00*)
		bSafeOUT_GT2_SafeDevOK : BOOL; (*SAFETY PLC: Gas safety device 2 OK*) (*OldName: new PV; Cycle: 5;*) (*V04.25.00.00*)
		bSafeOUT_GT3_SafeDevOK : BOOL; (*SAFETY PLC: Gas safety device 3 OK*) (*OldName: new PV; Cycle: 5;*) (*V04.25.00.00*)
		bSafeOUT_GT4_SafeDevOK : BOOL; (*SAFETY PLC: Gas safety device 4 OK*) (*OldName: new PV; Cycle: 5;*) (*V04.25.00.00*)
		bSafeOUT_DCGA_SafeDevOK : BOOL; (*SAFETY PLC: Gas safety device decentral gas addition OK*) (*OldName: new PV; Cycle: 5;*) (*V04.25.00.00*)
	END_STRUCT;
	MM2VIS_struct : 	STRUCT
		bEO_FreshOilPump : BOOL; (* *) (*OldName: NewPv V4.14*)
		bEO_WasteOilPump : BOOL; (* *) (*OldName: NewPv V4.14*)
		bEOVal_DemOpen : BOOL; (* *) (*OldName: NewPv V4.14*)
		bAct_Oil_Filling : BOOL; (*HMI SPARE  fresh oil pump start for oil filling*) (*OldName: NewPv V4.14*)
		bAct_Oil_Change : BOOL; (*HMI SPARE waste oil pump start for oil exchange*) (*OldName: NewPv V4.14*)
		bInitialOilFill_DemOpen : BOOL; (*Initial oil illing with engine oil valve*) (*OldName: NewPv V4.14*)
		bOilRefilOn : BOOL; (*Oil refilling with oil pump is on for the visualization*) (*OldName: NewPv V4.14*)
		rL_FreshOilTank : REAL; (*Tank fluid level measurement [mm] (or [l])*) (*OldName: NewPv V4.12*)
		rL_WasteOilTank : REAL; (*Tank fluid level measurement [mm] (or [l])*) (*OldName: NewPv V4.12*)
		rL_DayOilTank : REAL; (*Tank fluid level measurement [mm] (or [l])*) (*OldName: NewPv V4.12*)
		rV_FreshOilTank_Rel : REAL; (*Relative fluid level in tank, measured (calc.) [0-1]*) (*OldName: NewPv V4.12*)
		rV_WasteOilTank_Rel : REAL; (*Relative fluid level in tank, measured (calc.) [0-1]*) (*OldName: NewPv V4.12*)
		rV_DayOilTank_Rel : REAL; (*Relative fluid level in tank, measured (calc.) [0-1]*) (*OldName: NewPv V4.12*)
		rV_FreshOilTank : REAL; (*fluid volume in tank, measured /calculated [l]*) (*OldName: NewPv V4.12*)
		rV_WasteOilTank : REAL; (*fluid volume in tank, measured /calculated [l]*) (*OldName: NewPv V4.12*)
		rV_DayOilTank : REAL; (*fluid volume in tank, measured /calculated [l]*) (*OldName: NewPv V4.12*)
		rV_FreshOilTank_Max : REAL; (*total fluid volume in tank [l]*) (*OldName: NewPv V4.12*)
		rV_WasteOilTank_Max : REAL; (*total fluid volume in tank [l]*) (*OldName: NewPv V4.12*)
		rV_DayOilTank_Max : REAL; (*total fluid volume in tank [l]*) (*OldName: NewPv V4.12*)
		tCtr_CC_Out : _tGeACtrOut; (*crank case pressure controller*) (*OldName:new; Cycle:5*)
		tCtr_ECW_Out : _tGeACtrOut; (*engine cooling water controller*) (*OldName:new; Cycle:5*)
		rCtr_ECW_Set : REAL; (*engine cooling water temperature control valve setpoint[%]*) (*OldName:new; Cycle:5*)
		bTCOP_Dem : BOOL; (*turbo charger oil pump demand*) (*OldName:TLOP; Cycle:5*)
		rPr_CC : REAL; (*engine crank case pressure [bar]*) (*OldName: p_CC; Cycle:5*)
		bEOP1AC_Dem : BOOL; (*engine oil pump demand*) (*OldName:DO_EOP1AC; Cycle:5*)
		bEOP1DC_Dem : BOOL; (*engine oil pump demand*) (*OldName:DO_EOP1DC; Cycle:5*)
		bECWP1Dem : BOOL; (*engine cooling water pump demand*) (*OldName:B_SV[25]; Cycle:5*)
		bECWP2Dem : BOOL; (*engine cooling water pump demand*) (*OldName:A_MKWP2; Cycle:5*)
		bECWP_PreH_Dem : BOOL; (*engine cooling water preheating pump demand*) (*OldName:A_VORW; Cycle:5*)
		bECW_PreH_Dem : BOOL; (*engine cooling water preheating demand*) (*OldName:A_VORWH; Cycle:5*)
		bECW_PreHV_Opened : BOOL; (*engine cooling water preheating valve opened*) (*OldName:NVW1_O; Cycle:5*)
		bECW_CV_Open : BOOL; (*engine cooling water temp.control valve open*) (*OldName:TCV2_O; Cycle:5*)
		bMsg1017 : BOOL; (*Oil pressure low*) (*OldName:M_ODRA; Cycle:5*)
		bMsg1018 : BOOL; (*engine oil level low*) (*OldName:AMM_A10xx; Cycle:5*)
		bMsg1020 : BOOL; (*engine cooling water level low low*) (*OldName:AMM_A10xx; Cycle:5*)
		bMsg1023 : BOOL; (*engine startup failure*) (*OldName:AMM_A10xx; Cycle:5*)
		bMsg1043 : BOOL; (*Oil temperature high*) (*OldName:M_OTMA; Cycle:5*)
		bMsg1051 : BOOL; (*Engine oil level high*) (*OldName:M_OMAX; Cycle:5*)
		bMsg1052 : BOOL; (*gas pre alarm*) (*OldName:AMM_A10xx; Cycle:5*)
		bMsg1053 : BOOL; (*gas alarm*) (*OldName:AMM_A10xx; Cycle:5*)
		bMsg1054 : BOOL; (*fire alarm*) (*OldName:AMM_A10xx; Cycle:5*)
		bMsg1059 : BOOL; (*Oil filter differential pressure - Maximum*) (*OldName:_; Cycle:5*)
		bMsg1060 : BOOL; (*prelube oil pressure low*) (*OldName:AMM_A10xx; Cycle:5*)
		bMsg1090 : BOOL; (*engine cooling water pump failure*) (*OldName:AMM_A10xx; Cycle:5*)
		bMsg1091 : BOOL; (*charge cooling water pump failure*) (*OldName:AMM_A10xx; Cycle:5*)
		bMsg1100 : BOOL; (*water ingress into inlet manifold*) (*OldName:AMM_A11xx; Cycle:5*)
		bMsg1101 : BOOL; (*transformer failure*) (*OldName:AMM_A11xx; Cycle:5*)
		bMsg1120 : BOOL; (*speed measuring signal failure*) (*OldName:AMM_A11xx; Cycle:5*)
		bMsg1129 : BOOL; (*failure auxiliaries*) (*OldName:AMM_A11xx; Cycle:5*)
		bMsg1137 : BOOL; (*mains start device failure*) (*OldName:AMM_A11xx; Cycle:5*)
		bMsg1139 : BOOL; (*module control panel circuit breaker tripped*) (*OldName:AMM_W11xx; Cycle:5*)
		bMsg1140 : BOOL; (*interface control panel circuit breaker tripped*) (*OldName:AMM_W11xx; Cycle:5*)
		bMsg1148 : BOOL; (*Starter battery voltage low*) (*OldName:AMM_W11xx; Cycle:5*)
		bMsg1159 : BOOL; (*fresh oil tank level low*) (*OldName:AMM_W11xx; Cycle:5*)
		bMsg1160 : BOOL; (*waste oil tank level high*) (*OldName:AMM_W11xx; Cycle:5*)
		bMsg1166 : BOOL; (*Failure oil supply *) (*OldName:M_STOELV; Cycle:5*)
		bMsg1249 : BOOL; (*start engine on*) (*OldName:AMM_B12xx; Cycle:5*)
		bMsg1250 : BOOL; (*start engine off*) (*OldName:AMM_B12xx; Cycle:5*)
		bMsg1257 : BOOL; (*demand engine cooling water pump on*) (*OldName:NewPv; Cycle:5*)
		bMsg1258 : BOOL; (*demand engine cooling water pump off*) (*OldName:NewPv; Cycle:5*)
		bMsg1259 : BOOL; (*demand oil pump on*) (*OldName:NewPv; Cycle:5*)
		bMsg1260 : BOOL; (*demand oil pump off*) (*OldName:NewPv; Cycle:5*)
		bMsg1261 : BOOL; (*demand oil pump (DC) on*) (*OldName:NewPv; Cycle:5*)
		bMsg1262 : BOOL; (*demand oil pump (DC) off*) (*OldName:NewPv; Cycle:5*)
		bMsg1263 : BOOL; (*demand turbo charger oil pump on*) (*OldName:NewPv; Cycle:5*)
		bMsg1264 : BOOL; (*demand turbo charger oil pump off*) (*OldName:NewPv; Cycle:5*)
		bMsg1281 : BOOL; (*demand engine cooling water preheating pump on*) (*OldName:NewPv; Cycle:5*)
		bMsg1282 : BOOL; (*demand engine cooling water preheating pump off*) (*OldName:NewPv; Cycle:5*)
		bMsg1292 : BOOL; (*Manual operating auxiliaries control (Handbedienebene) active*) (*OldName:NewPv; Cycle:5*)
		bMsg2102 : BOOL; (*Engine oil temperature measuring signal failure*) (*OldName:pv; Cycle:5*)
		bMsg2103 : BOOL; (*Engine oil pressure measuring signal failure*) (*OldName:MS_ODR; Cycle:5*)
		bMsg2114 : BOOL; (*preheating pump failure*) (*OldName:AMM_W21xx; Cycle:5*)
		bMsg2118 : BOOL; (*failure charge cooler pump*) (*OldName:AMM_W21xx; Cycle:5*)
		bMsg2201 : BOOL; (*Engine turn equipment active*) (*OldName:AMM_A22xx; Cycle:5*)
		bMsg2213 : BOOL; (*Turbo charger oil filter differential pressure maximum*) (*OldName:pv; Cycle:5*)
		bMsg2224 : BOOL; (*measuring signal failure pressure after turbocharger oil filter*) (*OldName:pv; Cycle:5*)
		bMsg2233 : BOOL; (*pressure after turbocharger oil filter high*) (*OldName:bPv; Cycle:5*)
		bMsg2234 : BOOL; (*pressure after turbocharger oil filter low*) (*OldName:bPv; Cycle:5*)
		bMsg2238 : BOOL; (*Turbocharger pre-lube pressure low*) (*OldName:new; Cycle:5*)
		bMsg2242 : BOOL; (*Measuring signal failure oil pressure before oil filter*) (*OldName:MS_OELF; Cycle:5*)
		bMsg2260 : BOOL; (*Measuring signal failure oil pressure after oil filter*) (*OldName:pv; Cycle:5*)
		bMsg2263 : BOOL; (*preheating flap position signal failure*) (*OldName:AMM_A22xx; Cycle:5*)
		bMsg2264 : BOOL; (*engine cooling water pre heating temperature high*) (*OldName:AMM_A22xx; Cycle:5*)
		bMsg2265 : BOOL; (*engine oil preheating temperature high*) (*OldName:newPv; Cycle:5*)
		bMsg2266 : BOOL; (*startup failure hydraulic shock*) (*OldName:AMM_A22xx; Cycle:5*)
		bMsg2267 : BOOL; (*starter supply pressure high*) (*OldName:AMM_A22xx; Cycle:5*)
		bMsg2268 : BOOL; (*starter compressed air vessel pressure low*) (*OldName:AMM_A22xx; Cycle:5*)
		bMsg2269 : BOOL; (*air starter supply pressure low*) (*OldName:AMM_A22xx; Cycle:5*)
		bMsg2284 : BOOL; (*level engine oil sump high*) (*OldName:ALM[2284]; Cycle:5*)
		bMsg2291 : BOOL; (*engine oil pressure after pump high high M.03-PI-007*)
		bMsg2292 : BOOL; (*engine oil pressure after pump high safety pressure switch M.03-PS-001*)
		bMsg2304 : BOOL; (*Oil pressure before oil filter maximum, M.03-PI-002*)
		bMsg2332 : BOOL; (*boiler failure*)
		bMsg2333 : BOOL; (*seismic alarm M.00-AI-100*)
		bMsg2348 : BOOL; (*auxiliaries power supply circuit breaker module control panel tripped*)
		bMsg2349 : BOOL; (*auxiliaries power supply circuit breaker module control panel opened*)
		bMsg2350 : BOOL; (*Earth fault auxiliaries power supply module control panel*)
		bMsg2351 : BOOL; (*Earth fault frequency converter module control panel*)
		bMsg2352 : BOOL; (*Earth fault frequency converter module interface panel*)
		bMsg2353 : BOOL; (*Earth fault frequency converter auxiliaries control panel*)
		bMsg2355 : BOOL; (*Earth fault auxiliaries power supply auxiliaries control panel*)
		bMsg2359 : BOOL; (*auxiliaries power supply circuit breaker auxiliaries control panel tripped*)
		bMsg2360 : BOOL; (*auxiliaries power supply circuit breaker auxiliaries control panel opened*)
		bMsg2361 : BOOL; (*Leakage in additional external oil tank*) (*OldName:newPv; Cycle:5*)
		bMsg2376 : BOOL; (*Scavenging by starting system not succesful*)
		bMsg2377 : BOOL; (*Measuring signal failure voltage start motor 1*)
		bMsg2378 : BOOL; (*Measuring signal failure voltage start motor 2*)
		bMsg2379 : BOOL; (*Measuring signal failure voltage start motor 3*)
		bMsg2382 : BOOL; (*Start attempt failed minimum speed*)
		bMsg2421 : BOOL; (*Oil pressure before oil filter maximum, M.03-PI-002*)
		bMsg2422 : BOOL; (*Oil filter maintenance (oil filter unit) *)
		bMsg2423 : BOOL; (*engine oil preheating temperature high high*) (*SWAT920/1*)
		bMsg2424 : BOOL; (*Turning fly wheel during engagement*) (*SWAT920/2*)
		bMsg2425 : BOOL; (*air starter engaging error - no air pressure at pressure switch*) (*SWAT920/2*)
		bMsg2426 : BOOL; (*start speed pickup signal missing*) (*SWAT920/2*)
		bMsg2427 : BOOL; (*Engine oil pressure low - During permanent pre-lubrication or pre-heating *)
		bMsg2431 : BOOL; (*preheating flap position signal failure*) (*SWAT920/1*)
		bMsg2432 : BOOL; (*Measuring signal failure oil pressure after oil filter*) (*SWAT920/1*)
		bMsg2433 : BOOL; (*measuring signal failure pressure after turbocharger oil filter*) (*SWAT920/1*)
		bMsg2434 : BOOL; (*turbo charger oil pressure high - permanent prelubrication*)
		bMsg2435 : BOOL; (*engine oil level high*) (*SWAT920/2*)
		bMsg2459 : BOOL; (*measuring signal failure turbocharger oil pressure*)
		bMsg2473 : BOOL; (*starter battery voltage maximum*)
		bMsg2475 : BOOL; (*maintenance interval prelubrication pump*)
		bMsg2524 : BOOL; (*oil preheating temperature min / no start release*) (*OldName:bPv; Cycle:5*)
		bMsg2534 : BOOL; (*Oil filter differential pressure maximum --> NOT USED*) (*OldName:new; Cycle:5*)
		bMsg2545 : BOOL; (*startup failure starter --> NOT USED*) (*OldName:AMM_W25xx; Cycle:5*)
		bMsg2554 : BOOL; (*Pressure after turbocharger oil filter low*) (*OldName:bPv; Cycle:5*)
		bMsg2558 : BOOL; (*crank case pressure high*) (*OldName:AMM_W25xx; Cycle:5*)
		bMsg2557 : BOOL; (*measuring signal failure air starter supply pressure*)
		bMsg2559 : BOOL; (*measuring signal failure air starter tank pressure*)
		bMsg2560 : BOOL; (*starter compressed air vessel pressure low*) (*OldName:AMM_W25xx; Cycle:5*)
		bMsg2571 : BOOL; (*failure over voltage protection auxiliaries power supply*) (*OldName:AMM_W25xx; Cycle:5*)
		bMsg2572 : BOOL; (*failure uninterrupted power supply*) (*OldName:AMM_W25xx; Cycle:5*)
		bMsg2576 : BOOL; (*Measuring signal failure oilfill level*) (*OldName:pv; Cycle:5*)
		bMsg2579 : BOOL; (*Oilpressure min for oilpreheating*) (*OldName:ODR_VORW; Cycle:5*)
		bMsg2582 : BOOL; (*Pump switchover: cooldown oil pressure not achieved*) (*OldName:umschalt_NKUEHL; Cycle:5*)
		bMsg2587 : BOOL; (*signal failure oil quality sensor*) (*OldName:AMM_W25xx; Cycle:5*)
		bMsg2589 : BOOL; (*engine cooling water pre heating temperature high*) (*OldName:AMM_W25xx; Cycle:5*)
		bMsg2590 : BOOL; (*engine oil pre heating temperature high*) (*OldName:AMM_W25xx; Cycle:5*)
		bMsg2591 : BOOL; (*blowby fan speed high*) (*OldName:AMM_W25xx; Cycle:5*)
		bMsg2592 : BOOL; (*blowby fan speed low*) (*OldName:AMM_W25xx; Cycle:5*)
		bMsg2594 : BOOL; (*control voltage low - engine*) (*OldName:AMM_W25xx; Cycle:5*)
		bMsg2595 : BOOL; (*control voltage low - turbo charger aux.*) (*OldName:AMM_W25xx; Cycle:5*)
		bMsg2596 : BOOL; (*control voltage low - module control panel*) (*OldName:AMM_W25xx; Cycle:5*)
		bMsg2597 : BOOL; (*prelubrication pump failure - engine*) (*OldName:AMM_W25xx; Cycle:5*)
		bMsg2598 : BOOL; (*prelubrication pump turbo charger circuit breaker tripped*) (*OldName:AMM_W25xx; Cycle:5*)
		bMsg2599 : BOOL; (*prelubrication pump turbo charger USV circuit breaker tripped*) (*OldName:AMM_W25xx; Cycle:5*)
		bMsg2600 : BOOL; (*preheating pump circuit breaker tripped*) (*OldName:AMM_W26xx; Cycle:5*)
		bMsg2602 : BOOL; (*charging unit turbo charger auxiliaries circuit breaker tripped*) (*OldName:AMM_W26xx; Cycle:5*)
		bMsg2603 : BOOL; (*charging unit engine interface panel circuit breaker tripped*) (*OldName:AMM_W26xx; Cycle:5*)
		bMsg2604 : BOOL; (*power supply engine interface panel circuit breaker tripped*) (*OldName:AMM_W26xx; Cycle:5*)
		bMsg2605 : BOOL; (*control voltage transformer circuit breaker tripped*) (*OldName:AMM_W26xx; Cycle:5*)
		bMsg2606 : BOOL; (*service cooling water pump circuit breaker tripped*) (*OldName:AMM_W26xx; Cycle:5*)
		bMsg2608 : BOOL; (*engine AC prelubrication pump circuit breaker tripped*) (*OldName:AMM_W26xx; Cycle:5*)
		bMsg2613 : BOOL; (*oil pressure after TC oil filter high*) (*OldName:AMM_W26xx; Cycle:5*)
		bMsg2624 : BOOL; (*oil pressure LP TC A inlet*) (*OldName:AMM_W26xx; Cycle:5*)
		bMsg2625 : BOOL; (*oil pressure LP TC B inlet*) (*OldName:AMM_W26xx; Cycle:5*)
		bMsg2627 : BOOL; (*oil pressure before filter (oil filter unit) signal failure*) (*OldName:AMM_W26xx; Cycle:5*)
		bMsg2628 : BOOL; (*oil pressure after filter (oil filter unit) signal failure*) (*OldName:AMM_W26xx; Cycle:5*)
		bMsg2629 : BOOL; (*oil difference pressure filter (oil filter unit) high*) (*OldName:AMM_W26xx; Cycle:5*)
		bMsg2636 : BOOL; (*engine interface panel AC power supply circuit breaker tripped*) (*OldName:AMM_W26xx; Cycle:5*)
		bMsg2642 : BOOL; (*engine oil temperature oil pan signal failure*) (*OldName:AMM_W26xx; Cycle:5*)
		bMsg2643 : BOOL; (*oil temperature after pump signal failure*) (*OldName:AMM_W26xx; Cycle:5*)
		bMsg2644 : BOOL; (*UPS circuit breaker tripped*) (*OldName:AMM_W26xx; Cycle:5*)
		bMsg2645 : BOOL; (*engine interface panel power supply circuit breaker tripped*) (*OldName:AMM_W26xx; Cycle:5*)
		bMsg2646 : BOOL; (*engine interface panel UPS supply circuit breaker tripped*) (*OldName:AMM_W26xx; Cycle:5*)
		bMsg2648 : BOOL; (*measuring signal failure pressure before turbocharger oil filter*) (*OldName:AMM_W26xx; Cycle:5*)
		bMsg2649 : BOOL; (*W2649 Crank case pressure low  *)
		bMsg2650 : BOOL; (*W2650 Blow by blower not ready  *)
		bMsg2651 : BOOL; (*W2651 Measuring signal failure pressure before blow by filter  *)
		bMsg2652 : BOOL; (*W2652 Measuring signal failure pressure after blow by filter  *)
		bMsg2653 : BOOL; (*W2653 Blow by filter difference pressure high - maintenance  *)
		bMsg2654 : BOOL; (*W2654 Blow by filter difference pressure low  *)
		bMsg2666 : BOOL; (*preheating flap failure*) (*OldName:AMM_W26xx; Cycle:5*)
		bMsg2689 : BOOL; (*permanent prelibrication failure*) (*OldName:newPV; Cycle:5*)
		bMsg2722 : BOOL; (*fresh oil tank level high*) (*OldName:newPV; Cycle:5*)
		bMsg2723 : BOOL; (*overfill prevention device fresh oil tank tripped*) (*OldName:newPV; Cycle:5*)
		bMsg2724 : BOOL; (*leakage fresh oil tank*) (*OldName:newPV; Cycle:5*)
		bMsg2725 : BOOL; (*leakage fresh oil pump*) (*OldName:newPV; Cycle:5*)
		bMsg2726 : BOOL; (*overfill prevention device waste oil tank tripped*) (*OldName:newPV; Cycle:5*)
		bMsg2727 : BOOL; (*leakage waste oil tank*) (*OldName:newPV; Cycle:5*)
		bMsg2728 : BOOL; (*leakage waste oil pump*) (*OldName:newPV; Cycle:5*)
		bMsg2729 : BOOL; (*general failure oil system*) (*OldName:newPV; Cycle:5*)
		bMsg2737 : BOOL; (*Auxiliaries switch module interface tripped*) (*OldName:M_STOELV; Cycle:5*)
		bMsg2738 : BOOL; (*Release auxiliaries from auxiliaries panel is missing*) (*OldName:M_STOELV; Cycle:5*)
		bMsg2739 : BOOL; (*day oil tank maximum*) (*OldName:M_STOELV; Cycle:5*)
		bMsg2740 : BOOL; (*leckage day oil tnak*) (*OldName:M_STOELV; Cycle:5*)
		bMsg2741 : BOOL; (*day tank oil collector pan maximum*) (*OldName:M_STOELV; Cycle:5*)
		bMsg2742 : BOOL; (*auxiliaries switch module interface tripped*) (*OldName:M_STOELV; Cycle:5*)
		bMsg2754 : BOOL; (*Measuring signal failure pressure before blow by filter A*) (*OldName:newPv; Cycle:5*)
		bMsg2755 : BOOL; (*Measuring signal failure pressure before blow by filter B*) (*OldName:newPv; Cycle:5*)
		bMsg2756 : BOOL; (*Measuring signal failure pressure after blow by filter A*) (*OldName:newPv; Cycle:5*)
		bMsg2757 : BOOL; (*Measuring signal failure pressure after blow by filter B*) (*OldName:newPv; Cycle:5*)
		bMsg2758 : BOOL; (*differenzial pressure high blow by filter A - maintenance (*OldName:newPv; Cycle:5*)
		bMsg2759 : BOOL; (*differenzial pressure high blow by filter B - maintenance (*OldName:newPv; Cycle:5*)
		bMsg2760 : BOOL; (*differenzial pressure low blow by filter A*) (*OldName:newPv; Cycle:5*)
		bMsg2761 : BOOL; (*differenzial pressure low blow by filter B*) (*OldName:newPv; Cycle:5*)
		bMsg2762 : BOOL; (*plausibility check engine oil pressure*) (*OldName:newPv; Cycle:5*)
		bMsg2770 : BOOL; (*control voltage missing generator interface*) (*OldName:newPv;Cycle:5*)
		bMsg2771 : BOOL; (*control voltage missing engine interface bank B*) (*OldName:newPv;Cycle:5*)
		bMsg2772 : BOOL; (*control voltage missing turbo charger module interface *) (*OldName:newPv;Cycle:5*)
		bMsg2773 : BOOL; (*control voltage missing turbo charger unit sensor cabinet *) (*OldName:newPv;Cycle:5*)
		bMsg2774 : BOOL; (*control voltage missing jacket water module interface *) (*OldName:newPv;Cycle:5*)
		bMsg2775 : BOOL; (*control voltage missing oil module interface *) (*OldName:newPv;Cycle:5*)
		bMsg2776 : BOOL; (*control voltage missing module interface cabinet*) (*OldName:newPv;Cycle:5*)
		bMsg2777 : BOOL; (*control voltage missing module control cabinet *) (*OldName:newPv;Cycle:5*)
		bMsg2778 : BOOL; (*control voltage missing auxiliaries control cabinet1*) (*OldName:newPv;Cycle:5*)
		bMsg2781 : BOOL; (*control voltage missing auxiliaries control cabinet2*) (*OldName:newPv;Cycle:5*)
		bMsg2782 : BOOL; (*control voltage missing auxiliaries control cabinet3*) (*OldName:newPv;Cycle:5*)
		bMsg2783 : BOOL; (*control voltage missing auxiliaries control cabinet4*) (*OldName:newPv;Cycle:5*)
		bMsg2784 : BOOL; (*control voltage missing auxiliaries control cabinet5*) (*OldName:newPv;Cycle:5*)
		bMsg2785 : BOOL; (*Oil pressure before filter (oil filter unit) maximum*) (*OldName:new; Cycle:5*)
		bMsg2786 : BOOL; (*Oil pressure before centrifuge (oil filter unit) signal failure*) (*OldName:new; Cycle:5*)
		bMsg2787 : BOOL; (*Oil pressure before centrifuge (oil filter unit) maximum*) (*OldName:new; Cycle:5*)
		bMsg2788 : BOOL; (*Oil centrifuge interrupted power supply (oil filter unit)*) (*OldName:new; Cycle:5*)
		bMsg2789 : BOOL; (*Oil filter pump interrupted power supply (oil filter unit)*) (*OldName:new; Cycle:5*)
		bMsg2791 : BOOL; (*engine cooling water pump not ready*) (*OldName:newPv;Cycle:5*)
		bMsg2792 : BOOL; (*engine prelube oil pump not ready*) (*OldName:newPv;Cycle:5*)
		bMsg2809 : BOOL; (*preheating flap opened*) (*OldName:AMM_B28xx; Cycle:5*)
		bMsg2810 : BOOL; (*preheating flap closed*) (*OldName:AMM_B28xx; Cycle:5*)
		bMsg2931 : BOOL; (*Active Cooling Program in operation*)
		bMsg2932 : BOOL; (*Active Cooling Program finished*)
		bMsg2933 : BOOL; (*Active Cooling Program cancelled*)
		bMsg2956 : BOOL; (*Demand engine oil preheating valve open*)
		bMsg2957 : BOOL; (*Demand engine oil preheating valve close*)
		bMsg2978 : BOOL; (*Blow-by blower on*) (*OldName:newPv;Cycle:5*)
		bMsg2979 : BOOL; (*Blow-by blower off*) (*OldName:newPv;Cycle:5*)
		bMsg3216 : BOOL; (*Oil temperatur high*) (*OldName:M_OTMAW; Cycle:5*)
		bMsg3218 : BOOL; (*Oil pressure minimum*) (*OldName:M_ODRW; Cycle:5*)
		bMsg3300 : BOOL; (*blocking acknowledgement by starter temperature*) (*OldName:AT4_BLOCK; Cycle:5;*)
		bMsg3301 : BOOL; (*purge cycle - gas safety loop tripped*) (*OldName:AMM_A33xx; Cycle:5*)
		bMsg3304 : BOOL; (*Oil pressure low transmission*) (*OldName:pv; Cycle:5*)
		bMsg3305 : BOOL; (*Oil pressure high transmission*) (*OldName:pv; Cycle:5*)
		bMsg3322 : BOOL; (*crank case pressure high*) (*OldName:AMM_A33xx; Cycle:5*)
		bMsg3323 : BOOL; (*crank case pressure measuring signal failure*) (*OldName:AMM_A33xx; Cycle:5*)
		bMsg3350 : BOOL; (*CO alarm*) (*OldName:AMM_A33xx; Cycle:5*)
		bMsg3351 : BOOL; (*active filter alarm*) (*OldName:AMM_A33xx; Cycle:5*)
		bMsg3369 : BOOL; (*	Air starter supply pressure low*) (*OldName:newPv; Cycle:5*)
		bMsg3370 : BOOL; (*	Measuring signal failure air starter supply pressure*) (*OldName:newPv; Cycle:5*)
		bMsg3375 : BOOL; (*	Air starter engaging error*) (*OldName:newPv; Cycle:5*)
		bMsg3401 : BOOL; (*engine oil level low*) (*OldName:AMM_W34xx; Cycle:5*)
		bMsg3403 : BOOL; (*engine cooling water level low*) (*OldName:AMM_W34xx; Cycle:5*)
		bMsg3405 : BOOL; (*module control panel circuit breaker tripped*) (*OldName:AMM_W34xx; Cycle:5*)
		bMsg3413 : BOOL; (*Measuring signal failure oil pressure before oil filter --> NOT USED *) (*OldName:MS_OELF; Cycle:5*)
		bMsg3414 : BOOL; (*Oil filter differential pressure - Oil filter achieves service life limit*) (*OldName:bPv; Cycle:5*)
		bMsg3415 : BOOL; (*Oil filter differential pressure - Oil filter to be replaced*) (*OldName:bPv; Cycle:5*)
		bMsg3416 : BOOL; (*Oil filter differential pressure - Maximum --> NOT USED*) (*OldName:bPv; Cycle:5*)
		bMsg3495 : BOOL; (*engine oil pressure after pump high M.03-PI-007*)
		bMsg3496 : BOOL; (*engine oil pressure after pump signal failure M.03-PI-007*)
		bMsg3497 : BOOL; (*failure in the safety loop*) (*OldName:AMM_W34xx; Cycle:5*)
		bMsg3507 : BOOL; (*Oil pressure high*) (*OldName:M_ODR_MAX; Cycle:5*)
		bMsg3515 : BOOL; (*air conditioning unit failure in module interface panel*) (*OldName:AMM_W35xx; Cycle:5*)
		bMsg3519 : BOOL; (*heat water pump failure*) (*OldName:AMM_A35xx; Cycle:5*)
		bMsg3572 : BOOL; (*transformer failure*) (*OldName:AMM_W35xx; Cycle:5*)
		bMsg3574 : BOOL; (*active filter warning*) (*OldName:AMM_W35xx; Cycle:5*)
		bMsg3578 : BOOL; (*auxiliaries failure warning*) (*OldName:AMM_W35xx; Cycle:5*)
		bMsg3579 : BOOL; (*CO prealarm*) (*OldName:AMM_A33xx; Cycle:5*)
		bMsg3587 : BOOL; (*water ingress into inlet manifold*) (*OldName:AMM_W35xx; Cycle:5*)
		bMsg3588 : BOOL; (*inlet manifold fill sensor inactive*) (*OldName:AMM_W35xx; Cycle:5*)
		bMsg9001 : BOOL; (*Oil sample taken*)
		bMsg9002 : BOOL; (*Oil exchanged*)
		bMsg9003 : BOOL; (*Coolant sample taken*)
		bMsg9048 : BOOL; (*Coolant exchanged*)
		bMsg9067 : BOOL; (*Oil sampling interval extended*)
		bMsg9069 : BOOL; (*Buffer battery test in progress*)
		bMsg9070 : BOOL; (*Control battery test in progress*)
		bMsg9074 : BOOL; (*Tooth to tooth position*)
		bMsg9088 : BOOL; (*Scavenging by starting system successful*)
		bMsg9089 : BOOL; (*Starter motor 1 did not engage*)
		bMsg9090 : BOOL; (*Starter motor 2 did not engage*)
		bMsg9091 : BOOL; (*Starter motor 3 did not engage*)
		bMsg9096 : BOOL; (*Starter overheated*)
		bMsg9097 : BOOL; (*Purge cranking cycle initiated*)
		bMsg9214 : BOOL; (*engine turn equipment active, SWAT920/5*) (*OldName:; Cycle:5*)
		bMsg9220 : BOOL; (*plausibility check engine oil pressure after filter*) (*OldName:newPv; Cycle:5*)
		bMsg9221 : BOOL; (*pressure after turbocharger oil filter high - permanent prelubrification*)
		bMsg9222 : BOOL; (*Oil pressure after TC oil filter high - Permanent pre-lubrication or pre-heating OFF*)
		bMsg9224 : BOOL; (*engine oil pressure high - permanent prelubrification*)
		bMsg9225 : BOOL; (*Engine oil pressure high - Permanent pre-lubrication or pre-heating OFF*)
		bMsg9227 : BOOL; (*failure charge cooler 2 pump*) (*OldName:newPV; Cycle:5*)
		bMsg9254 : BOOL; (*Engine cooling water hydraulic pre-heating failure*) (*OldName:newPV; Cycle:5*)
		bMsg9255 : BOOL; (*Failure high temperature circuit pump 2 (redundant heating water pump)*) (*OldName:newPV; Cycle:5*)
		bMsg9256 : BOOL; (*Failure low temperature circuit pump 3 (redundant charge cooler pump)*) (*OldName:newPV; Cycle:5*)
		bMsg9257 : BOOL; (*Failure low temperature circuit pump 4 (redundant charge cooler 2 pump)*) (*OldName:newPV; Cycle:5*)
		bMsg9258 : BOOL; (*Failure emergency cooling circuit pump 2 (redundant emergency cooler pump)*) (*OldName:newPV; Cycle:5*)
		bMsg9279 : BOOL; (*Failure emergency cooling circuit pump 1 (emergency cooler pump)*) (*OldName:newPV; Cycle:5*)
		bMsg9280 : BOOL; (*Maximum number of failed post coolings for turbocharger exceeded; inspection of turbocharger required*)
		bMsg9281 : BOOL; (*Maximum number of failed post coolings for turbocharger at bank A exceeded; inspection of turbocharger required*)
		bMsg9282 : BOOL; (*Maximum number of failed post coolings for turbocharger at bank B exceeded; inspection of turbocharger required*)
		bMsg9283 : BOOL; (*Failed post cooling for turbocharger detected*)
		bMsg9303 : BOOL; (*Measuring signal failure air starter engagement pressure*)
		bMsg9314 : BOOL; (*Engine cooling water pump circuit breaker tripped*)
		bMsg9316 : BOOL; (*Measuring signal failure cooling water pressure after ECW pump 1*)
		bMsg9317 : BOOL; (*Measuring signal failure cooling water pressure after ECW pump 2*)
		bMsg9322 : BOOL; (*Fresh oil tank level low (2nd level switch)*)
		bMsg9323 : BOOL; (*Fresh oil day tank level low*)
		bMsg9324 : BOOL; (*Fresh oil day tank level low (2nd level switch)*)
		bMsg9325 : BOOL; (*Overfill prevention device fresh oil day tank tripped*)
		bMsg9326 : BOOL; (*Waste oil day tank level high*)
		bMsg9327 : BOOL; (*Overfill prevention device waste oil day tank tripped*)
		bMsg9328 : BOOL; (*Fresh oil pump oil pressure maximum*)
		bMsg9332 : BOOL; (*Take oil sample*)
		bMsg9333 : BOOL; (*Take coolant sample*)
		bMsg9334 : BOOL; (*Buffer battery 1 voltage low*)
		bMsg9335 : BOOL; (*Buffer battery 2 voltage low*)
		bMsg9336 : BOOL; (*Battery charging device malfunction*)
		bMsg9352 : BOOL; (*Oil quality sensor: Measurement signal failure, return to regular sampling interval*)
		bMsg9353 : BOOL; (*Oil quality sensor: Oil quality warning, return to regular sampling interval*)
		bMsg9354 : BOOL; (*Oil quality sensor: Critical oil quality warning, return to regular sampling interval*)
		bMsg9355 : BOOL; (*Oil quality sensor: Increased oil aging, return to regular sampling interval*)
		bMsg9356 : BOOL; (*Oil quality sensor: Critical oil aging, return to regular sampling interval*)
		bMsg9357 : BOOL; (*Control battery voltage low*)
		bMsg9358 : BOOL; (*Control battery charging device malfunction*)
		bMsg9359 : BOOL; (*Oil pressure before centrifuge (oil filter unit) minimum*)
		bMsg9362 : BOOL; (*Fresh Oil tank Monitoring sensor signal failure *) (*OldName: new variable V4.12; Cyclic 5*)
		bMsg9363 : BOOL; (*Waste Oil tank Monitoring sensor signal failure *) (*OldName: new variable V4.12; Cyclic 5*)
		bMsg9364 : BOOL; (*Day Oil tank Monitoring sensor signal failure *) (*OldName: new variable V4.12; Cyclic 5*)
		bMsg9369 : BOOL; (*W9369 Failure auxiliaries supply voltage engine *) (*OldName: new variable V4.12; Cyclic 5*)
		bMsg9378 : BOOL; (*Oil refill volume maximum*) (*OldName:new variable; Cycle:5*) (*V04.13.00.00*)
		bMsg9390 : BOOL; (*Oil temperature before engine start too low*) (*OldName:new variable; Cycle:5*) (*V04.13.00.00*)
		bMsg9435 : BOOL; (*Fire detection system - System failure*) (*SAFETY PLC*) (*V04.25.00.00*)
		bMsg9436 : BOOL; (*Gas detection system - System failure*) (*SAFETY PLC*) (*V04.25.00.00*)
		bMsg9513 : BOOL; (*Engine oil refilling failure*) (*2024-225*)
		bMsg9560 : BOOL; (*Fire detection system - System failure*) (*SAFETY PLC*) (*V04.25.00.00*)
		bMsg9561 : BOOL; (*Gas detection system - System failure*) (*SAFETY PLC*) (*V04.25.00.00*)
		rOC_Consum_Avg : REAL; (*Oil volume average (depends on Avg check box on VISU)*) (*OldName:new variable; Cycle:5*)
		rOC_Energy_Avg : REAL; (*Active energy average (depends on Avg check box on VISU)*) (*Active energy average  (*OldName:rAvgActiveEnergy; Cycle:5*)
		rVol_OC_Avg : REAL; (*Oil volume average (depends on Avg check box on VISU)*) (*Oil volume average  (*OldName:rAvgOilVolume; Cycle:5*)
		rP_OC_Energy : REAL; (*EO_Cnt trending: active energy during last measurement*) (*OldName:slActiveEnergy; Cycle:5*)
		rP_OC_Avg : REAL; (*EO_Cnt trending: average power during the measurement*) (*OldName:slAvgPower; Cycle:5*)
		rOC_DeltaOpHour : REAL; (*EO_Cnt trending: operating hours during last measurement*) (*OldName:slDeltaBh; Cycle:5*)
		rOC_Consum : REAL; (*EO_Cnt trending: oil consumption during during last measurement *) (*OldName:eOilConsumption; Cycle:5*)
		rVol_OC : REAL; (*EO_Cnt trending: oil volume during last measurement *) (*OldName:ssOilVolume; Cycle:5*)
		bEOF_PreheatRel : BOOL; (*DO: Release oil preheating valve *) (*OldName:new; Cycle:5*)
		bEO_Preheat1 : BOOL; (*DO: engine oil preheating element 1*) (*OldName:new; Cycle:5*)
		bEO_Preheat2 : BOOL; (*DO: engine oil preheating element 2*) (*OldName:new; Cycle:5*)
		bEO_Preheat3 : BOOL; (*DO: engine oil preheating element 3*) (*OldName:new; Cycle:5*)
		rEO_Level : REAL; (*Oil fill level*) (*OldName:OilFill; Cycle:5*)
		rPr_EO_diff_f : REAL; (*Calculation for Motor Oil filter pressure difference*) (*OldName:OilPress_diff_f; Cycle:5*)
		rPr_EOF_DiffMon : REAL; (*Oil pressure before oil filter *) (*OldName:ssOilPbFilter; Cycle:5*)
		rPr_EOF_Diff : REAL; (*engine oil filter pressure difference(before/last point)*) (*OldName:ssOilFilterPress; Cycle:5*)
		rPr_EngLubOil : REAL; (*Pressure engine lube oil [bar]*) (*OldName:ANA.ODR; Cycle:5*)
		tEO_Counter : ARRAY[0..19]OF tOilCounter; (*Circular buffer*) (*OldName:new; Cycle:5*)
		tCtr_EOVal_Out : _tGeACtrOut; (*engine oil cooler valve controller*) (*OldName:new; Cycle:5*)
		tCtr_EOVal_LT_Out : _tGeACtrOut; (*engine oil cooler LT valve controller*) (*OldName:new; Cycle:5*)
		rPr_EOF_After : REAL; (*Engine oil pressure after oil filter, NUP57/ M.03-PI-057*) (*OldName:OilPress_a_f; Cycle:5*)
		rPr_TC_EOF_After : REAL; (*Oil pressure after turbocharger oil filter, J920: NUP62/ M.03-PI-062 // J6: M.03-PI-063*) (*OldName:OilPress_a_ATL_f; Cycle:5*)
		rPr_TC_EOF_Before : REAL; (*Oil pressure in front of turbocharger oil filter, NUP61/ M.03-PI-061*) (*OldName:OilPress_f_ATL_f; Cycle:5*)
		rT_EO : REAL; (*Oil temperature*) (*OldName:ANA.OTP; Cycle:5*)
		rT_EOP_After : REAL; (*Oiltemperature after oilpump, NUT71/ M.03-TI-071*) (*OldName:OilTemp_a_op; Cycle:5*)
		bEng_StaSpdExc : BOOL; (*engine starter speed exceeded*) (*OldName:M_DREHZ; Cycle:5*)
		bTC_EOP_On : BOOL; (*turbo charger oil pump on*) (*OldName:TLOP; Cycle:5*)
		rTi_EngStart_Max : REAL; (*calculated max. allowed automatic start time (pilot)*) (*OldName:new; Cycle:5*)
		rN_EngStart : REAL; (*measured reference speed at last start after 5sec cranking (pilot)*) (*OldName:new; Cycle:5*)
		rTi_EngStart_Duration : REAL; (*actual automatic start time of the last start atemp (pilot)*)
		rTi_EngStart_Delay : REAL; (*actual automatic start time pause until the next start atemp (pilot)*)
		rT_EO_Pan : REAL; (*engine oil temperature oil pan, M.03-TI-002*) (*OldName:t_OilPan; Cycle:5*)
		rT_EO_Preheating : REAL; (*oil temperature preheating NUT78/ M.03-TI-078*) (*OldName:OilTemp_preh; Cycle:5*)
		rPr_Oil_LPTC_In_A : REAL; (*oil pressure LP turbo charger A inlet*) (*OldName:p_Oil_LPTC_InA; Cycle:5;*)
		rPr_Oil_LPTC_In_B : REAL; (*oil pressure LP turbo charger B inlet*) (*OldName:p_Oil_LPTC_InB; Cycle:5;*)
		rPr_f_BbFilt : REAL; (*Pressure before Blow-by filter [bar]*) (* Oldname: newPV, Cycle:5 *)
		rPr_f_BbFilt_A : REAL; (*Pressure before Blow-by filter A [bar]*) (* Oldname: newPV, Cycle:5 *)
		rPr_f_BbFilt_B : REAL; (*Pressure before Blow-by filter B [bar]*) (* Oldname: newPV, Cycle:5 *)
		rPr_a_BbFilt : REAL; (*Pressure after Blow-by filter [bar]*) (* Oldname: newPV , Cycle:5 *)
		rPr_a_BbFilt_A : REAL; (*Pressure after Blow-by filter A [bar]*) (* Oldname: newPV , Cycle:5 *)
		rPr_a_BbFilt_B : REAL; (*Pressure after Blow-by filter B [bar]*) (* Oldname: newPV , Cycle:5 *)
		rDPr_BbFilt : REAL; (*calculated blow-by filter difference pressure*) (* Oldname: newPV , Cycle:5 *)
		rDPr_BbFilt_A : REAL; (*calculated blow-by filter difference pressure bank A*) (* Oldname: newPV , Cycle:5 *)
		rDPr_BbFilt_B : REAL; (*calculated blow-by filter difference pressure bank B*) (* Oldname: newPV , Cycle:5 *)
		rPr_AirStarter_Tank : REAL; (*AI air starter tank pressure [bar] (P.31-PI-001)*) (* Oldname:newPV , Cycle:5 *)
		rPr_AirStarter_Supply : REAL; (*Air starter supply pressure [bar] (E.31-PI-001)*) (* Oldname:newPV , Cycle:5 *)
		rN_AirStarter : REAL; (*AI (Counter Modul) air starter speed [rpm] (E.00-SI-006)*) (* Oldname:newPV , Cycle:5 *)
		bManOpAuxCtr_Gnl_Rel : BOOL; (*General release. Safety conditions (gas alarm, fire alarm, safety loop, ..) are OK.*) (*OldName: newPV; Cycle: 5;*)
		rPr_EOaP : REAL; (*engine oil pressure after pump M.03-PI-007*) (* Oldname:newPV;Cycle:5*)
		rPr_OFUbFilt : REAL; (*pressure oil filter unit before filter M.03-PI-011*) (*OldName:newPV;Cycle:5*)
		rPr_OFUaFilt : REAL; (*pressure oil filter unit after filter M.03-PI-012*) (*OldName:newPV;Cycle:5*)
		rDPr_OFU_Filt : REAL; (*filter difference pressure oil filter unit M.03-PI-012*) (*OldName:newPV;Cycle:5*)
		rPr_OFUbCentrifuge : REAL; (*pressure oil filter unit before centrifuge M.03-PI-008 [bar]*) (* Oldname:new PV , Cycle:5 *)
		bOFUP_Centrifuge : BOOL; (*oil filter unit pump centrifuge M.03-P-006*) (*OldName:newPV;Cycle:5*)
		bOFUP_Filter : BOOL; (*oil filter unit pump filter M.03-P-007*) (*OldName:newPV;Cycle:5*)
		bTCOV_CoClose : BOOL; (*TC oil valve command close M.03-YCS-003*)
		rPr_TCO : REAL; (*pressure oil before turbo charger M.03-PI-063*)
		rU_StarterBat : REAL; (*starter battery voltage monitoring*)
		bPreL_FS_EngStaRel : BOOL; (*prelubrication engine fast start release*) (* Oldname:newPV;Cycle:5*)
		bRelEngOp_Aux : BOOL; (* release engine operation from auxiliaries with dropout delay *)
		bECW_HydrPreH_Dem : BOOL; (*Hydraulic ECW pre-heating demand*)
		rT_HW_Su_PreH_ECW_LimLo : REAL; (*Heating water temperature supply hydraulic ECW preheating limit low [°C]*)
		rT_HW_Su_PreH_ECW_LimHi : REAL; (*Heating water temperature supply hydraulic ECW preheating limit high [°C]*)
		bHWP1_Op : BOOL; (*Redundant heating water pump 1 operating (P.06-M-001)*)
		bHWP2_Op : BOOL; (*Redundant heating water pump 2 operating (P.06-M-002)*)
		bCCWP1_Op : BOOL; (*Redundant charge cooler water pump 1 operating (P.07-M-003)*)
		bCCWP2_Op : BOOL; (*Redundant charge cooler water pump 2 operating (P.07-M-013)*)
		bCC2WP1_Op : BOOL; (*Redundant charge cooler 2 water pump 1 operating (P.07-M-007)*)
		bCC2WP2_Op : BOOL; (*Redundant charge cooler 2 water pump 2 operating (P.07-M-017)*)
		bEmCWP1_Op : BOOL; (*Redundant emergency cooler water pump 1 operating (P.09-M-001)*)
		bEmCWP2_Op : BOOL; (*Redundant emergency cooler water pump 2 operating (P.09-M-002)*)
		rPr_AirST_Engage : REAL; (*Pressure air starter engagement [bar] (E.31-PI-004)*)
		bAirST_ValEngage : BOOL; (*Command air starter engagement valve (E.31-YCS-001)*)
		bAirST_ValStart : BOOL; (*Command air starter start valve (E.31-YCS-002)*)
		rPr_ECWaP1 : REAL; (*AI Engine cooling water pressure after ECW pump 1 (M.04-PI-010)*)
		rPr_ECWaP2 : REAL; (*AI Engine cooling water pressure after ECW pump 2 (M.04-PI-011)*)
		bHorn_Active : BOOL; (*Horn output active bit for visibility of horn off button*)
		iCnt_OilOh : DINT; (*Oil operating hours [Oh]*)
		iCnt_OilSampleOh : DINT; (*Oil operating hours until next sample [Oh]*)
		tLastOilExchange : tFluidEvent; (*operating data at last oil exchange*)
		tLastOilSample : tFluidEvent; (*Last oil sample information*)
		iCnt_CWOh : DINT; (*Cooling water operating hours [Oh]*)
		iCnt_CWSampleOh : DINT; (*Cooling water operating hours until next sample [Oh]*)
		tLastCWExchange : tFluidEvent; (*Last cooling water exchange information*)
		tLastCWSample : tFluidEvent; (*Last cooling water sample information*)
		bNoExtendedPrelube : BOOL; (*No extended prelubrication active (allows 5min start)*)
		rU_BufferBat1 : REAL; (*AI Buffer battery 1 voltage*)
		rU_BufferBat2 : REAL; (*AI Buffer battery 2 voltage*)
		rU_StarterBat_BatTest : REAL; (*Starter battery voltage last measurement*)
		rU_BufferBat1_BatTest : REAL; (*Buffer battery 1 voltage last measurement*)
		rU_BufferBat2_BatTest : REAL; (*Buffer battery 2 voltage last measurement*)
		bBatMon_TestRunning : BOOL; (*Status battery test*)
		iLeak_OilExtensionTank : INT; (*Oil leakage affected additional oil tank - HMI assistant value for alarm A2361*)
		rU_CtrlBat : ARRAY[1..iNum_CtrlBatMon]OF REAL; (*AI Control battery voltage*)
		rU_CtrlBat_BatTest : ARRAY[1..iNum_CtrlBatMon]OF REAL; (*Control battery voltage last measurement*)
		bCtrlBatMon_TestRunning : BOOL; (*Status battery test*)
		iNumActive_CtrlBatMon : USINT; (*Nr of active control battery test sets*)
		sLocIdent_CtrlBatMon : ARRAY[1..iNum_CtrlBatMon]OF STRING[10]; (*Control battery test set location*)
		sCtrlBat_LocFault : STRING[10]; (*Location of faulty control battery*)
		sCtrlBat_ChargeDev_LocFault : STRING[10]; (*Location of faulty control battery charging device*)
		bCtrlBat_Used : ARRAY[1..iNum_CtrlBatMon]OF BOOL; (*Control battery set [x] using*)
		bCtrlBat_UnderTest : ARRAY[1..iNum_CtrlBatMon]OF BOOL; (*Control battery set [x] under testing*)
		bBufferBat_UnderTest : ARRAY[1..iNum_CtrlBatMon]OF BOOL; (*Buffer battery set [x] under testing*)
		bStarterBat_UnderTest : BOOL; (*Starter battery under testing*)
		bU_StarterBat_Exist : BOOL; (*Starter battery voltage exists*)
		rT_Oil_OQS_OC : REAL; (*Oil quality sensor: oil temperature*)
		rT_Sensor_OQS_OC : REAL; (*Oil quality sensor: sensor temperature*)
		rOilCond_OQS_OC_Unfilt : REAL; (*Oil quality sensor: oil condition value unfiltered*)
		rOilQual_OQS_OC : REAL; (*Oil quality sensor: oil quality*)
		rOilQual_OQS_OC_Unfilt : REAL; (*Oil quality sensor: oil quality unfiltered*)
		rOilQualTendency_OQS_OC : REAL; (*Oil quality sensor: oil quality tendency*)
		iOQS_OC_Status : INT; (*Oil quality sensor: Oil quality status*)
		iOQS_OC_Status_Num : INT; (*Oil quality sensor: Oil quality numerical status*)
		iOQS_OilSampleOh : DINT; (*Oil quality sensor: Recommended oil sampling interval*)
		iOQS_OC_OilTypeIdx : UINT; (*Oil quality sensor: oil type active*)
		bHWP_On : BOOL; (*Heating water pump ON*)
		bU_Starter_engage1 : BOOL; (*Start motor 1 function voltage GoodQual*)
		iVol_PurgeAir : UDINT; (*Volume of purge air [lt]*)
		bSt_Purge : BOOL; (*Purge state (true: engine purged, false: engine not purged)*)
		bFS_Rdy_STT_StPurge : BOOL; (*purge state and starter temperature readiness for fast start*)
		iNum_Msg9096 : DINT; (*B9096 starter overheated duration until release [s]*)
		iTi_ST_Res : UDINT; (*remaining starting time [s]*)
	END_STRUCT;
	OUT_AG_struct : 	STRUCT
		tEO_FreshOilPump_Dem : HALioDo_Type; (*fresh oil pump*) (*OldName:new V4.14; Cycle:5*)
		tEO_WasteOilPump_Dem : HALioDo_Type; (*waste oil pump*) (*OldName:new V4.14; Cycle:5*)
		bAux_OilValve_IsOpen : BOOL; (*valve status for fresh/waste oil in oil pan (without TOF), to be used for release of customized oil pump controls*) (*OldName:new V4.14; Cycle:5*)
		iIdx_ProcessStep_AG : DINT; (*Optional step information to display on VIS*) (*New 2016*)
		iProcessStepTime_AG : DINT; (*Optional step time  info to display on VIS*) (*New 2016*)
		tFreshOilPump_RTC : HALioDo_Type; (*fresh oil pump run time exceeded*) (*OldName:new; Cycle:5*)
		tCDP_Dem : HALioDo_Type; (*demand condensor pump*) (*OldName:new; Cycle:5*)
		rP_Red_TransformerWarning_Norm : REAL; (*Transformer power reduction setpoint*) (*OldName:new; Cycle:5*)
		bP_Red_TransformerWarning_Sel : BOOL; (*Transformer power reduction active*) (*OldName:new; Cycle:5*)
		tAG2AB : MM2AmmBase; (*MM2AmmBase*) (*OldName:new; Cycle:5*)
		tAG2PB : MM2ParaBase_type; (*MM2ParaBase*) (*OldName:new; Cycle:5*)
		bMsg1023 : BOOL; (*engine startup failure*) (*OldName:M_ANSTAN; Cycle:5*)
		bMsg1052 : BOOL; (*gas pre alarm*) (*OldName:M_GALV; Cycle:5*)
		bMsg1053 : BOOL; (*gas alarm*) (*OldName:M_GAL; Cycle:5*)
		bMsg1054 : BOOL; (*fire alarm*) (*OldName:M_BAL; Cycle:5*)
		bMsg1060 : BOOL; (*prelube oil pressure low*) (*OldName:M_VSD; Cycle:5*)
		bMsg1120 : BOOL; (*speed measuring signal failure*) (*OldName:AMM_A11xx; Cycle:5*) (*V04.01.00.00*)
		bMsg2102 : BOOL; (*engine oil temperature measuring signal failure*) (*OldName:M_MSODR; Cycle:5;*)
		bMsg2103 : BOOL; (*engine oil pressure measuring signal failure*) (*OldName:M_MSOTP; Cycle:5;*)
		bMsg2524 : BOOL; (*engine oil preheating temperature min / no start release*) (*OldName:newPV; Cycle:5;*)
		bMsg9214 : BOOL; (*Engine turn equipment active, SWAT920/5*) (*OldName:; Cycle:5*)
		bEngAutStartDelay : BOOL; (*engine automatic start delay*) (*OldName:AT3; Cycle:5*)
		bRelEngOp_Aux : BOOL; (* release engine operation from auxiliaries with dropout delay *) (*OldName:T6; Cycle:5*)
		bEngAuxMon : BOOL; (* engine auxiliaries monitoring *) (*OldName:ZM_HBT_UW; Cycle:5*)
		bEngOilLevel_Lo : BOOL; (* engine oil level low *) (*OldName:ZM_OMIN; Cycle:5*)
		bEngOilLevel_W_Lo : BOOL; (* engine oil level low warning SWAT#3 *) (*OldName: newPV; Cycle:5*)
		bEOP_AC_PowSupOk : BOOL; (* engine oil pump AC power supply ok *) (*OldName:SPG_VSP; Cycle:5*)
		bEng_Start : BOOL; (*engine start*) (*OldName:M_STRT; Cycle:5*)
		bJmpPLTime : BOOL; (* jump prelubrication time in case of emergency power supply *) (*OldName:UB_VORS; Cycle:5*)
		bLockAckStarter : BOOL; (* lockout acknowledgement by starter temperature *) (*OldName:AT4_BLOCK; Cycle:5*)
		bMaxPreLubeTime : BOOL; (* maximum engine prelubrication time *) (*OldName:T86; Cycle:5*)
		bRel_IgnOn : BOOL; (* release ignition ON *) (*OldName:AT5; Cycle:5*)
		bGV_Start_ScaveBlock : BOOL; (*block gas valves from startup procedure*)
		tAuxPoSuMains : HALioDo_Type; (*DO auxiliaries power supply from mains *) (*OldName:SPG_N; Cycle:5*)
		tAuxPoSuUPS : HALioDo_Type; (*DO auxiliaries power supply from UPS *) (*OldName:SPG_W; Cycle:5*)
		tChargeOff_Dem : HALioDo_Type; (*DO charging unit off demand*) (*OldName:CH_OFF; Cycle:5*)
		tECW_PreH_Dem : HALioDo_Type; (*DO engine cooling water preheating demand *) (*OldName:A_VORWH; Cycle:5*)
		tECW_PreH1Dem : HALioDo_Type; (*DO engine cooling water preheating 1 demand *) (*OldName:NHW101; Cycle:5*)
		tECW_PreH2Dem : HALioDo_Type; (*DO engine cooling water preheating 2 demand *) (*OldName:NHW102; Cycle:5*)
		tECW_PreH3Dem : HALioDo_Type; (*DO engine cooling water preheating 3 demand *) (*OldName:NHW103; Cycle:5*)
		tECWP_PreH_Dem : HALioDo_Type; (*DO engine cooling water preheating pump demand *) (*OldName:A_VORW; Cycle:5*)
		tECWP1Dem : HALioDo_Type; (*DO engine cooling water pump 1 demand *) (*OldName:A_MKWP; Cycle:5*)
		tECWP2Dem : HALioDo_Type; (*DO engine cooling water pump 2 demand *) (*OldName:A_MKWP2; Cycle:5*)
		tECW_PreHV_CoClose : HALioDo_Type; (*DO engine cooling water preheating valve - command close *) (*OldName:VORW_NVW1_C; Cycle:5*)
		tECW_PreHV_CoOpen : HALioDo_Type; (*DO engine cooling water preheating valve - command open *) (*OldName:VORW_NVW1_O; Cycle:5*)
		tEleStarter_Dem : HALioDo_Type; (*DO electric starter demand *) (*OldName:A_STRT; Cycle:5*)
		tEOP1AC_Dem : HALioDo_Type; (*DO engine oil pump 1 AC (M.03-P-002)*) (*OldName:DO_EOP1AC; Cycle:5*)
		tEOP1DC_Dem : HALioDo_Type; (*DO engine oil pump 1 DC (M.03-P-003)*) (*OldName:DO_EOP1DC; Cycle:5*)
		tEOVal_DemOpen : HALioDo_Type; (*DO engine oil refill valve demand open *) (*OldName:OELV_AUF; Cycle:5*)
		tHorn : HALioDo_Type; (*DO horn  *) (*OldName:HUPE; Cycle:5*)
		tHorn_Trip : HALioDo_Type; (*DO horn engine shutdown *) (*OldName:HUPE_A; Cycle:5*)
		tHorn_Warning : HALioDo_Type; (*DO horn warning *) (*OldName:HUPE_W; Cycle:5*)
		tHWP_Dem : HALioDo_Type; (*DO heating water pump demand (P.06-M-001)*) (*OldName:ANF_HWP; Cycle:5*)
		tMainGV_Rel : HALioDo_Type; (*DO main gas valve release *) (*OldName:FG_HGV; Cycle:5*)
		tMainsStartDevDem : HALioDo_Type; (*DO mains start device demand *) (*OldName:ANF_NST; Cycle:5*)
		tN_ECWP_Set : HALioAo_Type; (*AO speed engine cooling water pump setpoint*) (*OldName:setpoint_mkw_prom; Cycle:5*)
		tRotatingLight : HALioDo_Type; (*DO rotating light yellow *) (*OldName:ROLL; Cycle:5*)
		tSignal1R1 : HALioDo_Type; (*DO signal lamp 1 red continuous light *) (*OldName:DO_Signal1R1; Cycle:5*)
		tSignal1R2 : HALioDo_Type; (*DO signal lamp 2 red continuous light *) (*OldName:DO_Signal1R2; Cycle:5*)
		tSignalG1 : HALioDo_Type; (*DO signal lamp 1 green continuous light *) (*OldName:DO_SignalG1; Cycle:5*)
		tSignalG2 : HALioDo_Type; (*DO signal lamp 2 green continuous light *) (*OldName:DO_SignalG2; Cycle:5*)
		tSignalR1 : HALioDo_Type; (*DO signal lamp 1 red flashing *) (*OldName:DO_SignalR1; Cycle:5*)
		tSignalR2 : HALioDo_Type; (*DO signal lamp 2 red flashing *) (*OldName:DO_SignalR2; Cycle:5*)
		tSignalY1 : HALioDo_Type; (*DO signal lamp 1 yellow continuous light *) (*OldName:DO_SignalY1; Cycle:5*)
		tSignalY2 : HALioDo_Type; (*DO signal lamp 2 yellow continuous light *) (*OldName:DO_SignalY2; Cycle:5*)
		tStUpSpeed : HALioDo_Type; (*DO startup speed *) (*OldName:new; Cycle:5*)
		tTurnRel : HALioDo_Type; (*DO crank shaft turning device release*) (*OldName:FG_TURN; Cycle:5*)
		tCtr_ECW_Set : HALioAo_Type; (*AO engine cooling water temp.control valve setpoint*) (*OldName:TCV2_y; Cycle:5*)
		rPr_EO_CalcLim : REAL; (*Calculated oil pressure limit*) (*OldName:EGW_ODRA; Cycle:5;*)
		rPr_EO_Min : REAL; (*Oil pressure minimum*) (*OldName:GW_ODRA; Cycle:5;*)
		bPr_EOP_Prelub1 : BOOL; (*Prelubrication pressure 1 pump*) (*OldName:AN_VSD1; Cycle:5;*)
		bPr_EOP_Prelub2 : BOOL; (*Prelubrication pressure 2 pumps*) (*OldName:AN_VSD2; Cycle:5;*)
		bPr_EOP_MonActive : BOOL; (*Activation oil pressure monitoring*) (*OldName:M_DR_ODR; Cycle:5;*)
		tTC_EOP_On : HALioDo_Type; (*DO: Engine oil pump, NPO601*) (*OldName:TL_OP; Cycle:5;*)
		tTC_EOP_OnUSV : HALioDo_Type; (*DO: Engine oil pump, NPO601 via USV*) (*OldName:TL_OP_USV; Cycle:5;*)
		tEOP_On : HALioDo_Type; (*DO: Engine oil pump, NPO602*) (*OldName:M_OP; Cycle:5;*)
		bT_EO_PrehStartRel : BOOL; (*Release engine start from oil preheating temperature*) (*OldName:OIL_STARTFG; Cycle:5;*)
		tEO_Preheat1 : HALioDo_Type; (*DO: engine oil preheating element 1*) (*OldName:OIL_VORWH1; Cycle:5;*)
		tEO_Preheat2 : HALioDo_Type; (*DO: engine oil preheating element 2*) (*OldName:OIL_VORWH2; Cycle:5;*)
		tEO_Preheat3 : HALioDo_Type; (*DO: engine oil preheating element 3*) (*OldName:OIL_VORWH3; Cycle:5;*)
		tEOP_FC_Set : HALioAo_Type; (*AO: Setpoint frequency converter motor oil pump prelubrication, [100% = 1.0]*) (*OldName:setpoint_oilpump; Cycle:5;*)
		rP_Red_T_Oil_Norm : REAL; (*power reduction by oil temp. max related to rP_Nom*) (*OldName:RED_OLT; Cycle:5;*)
		tOV_Ctrl_Set : HALioAo_Type; (*AO: engine oil cooler setpoint*) (*OldName:AO_EOC_HT_sp; Cycle:5;*)
		tEOVal_LT_Set : HALioAo_Type; (*AO: engine oil cooler LT setpoint*) (*OldName:AO_EOC_LT_sp; Cycle:5;*)
		bT_EOP_RelLoad : BOOL; (*Oil temperature release load*) (*OldName:OT_LFG; Cycle:5;*)
		tEOF_PreheatRel : HALioDo_Type; (*DO: Release oil preheating valve *) (*OldName:OILVORW_SOV; Cycle:5;*)
		tBbBlower_y : HALioAo_Type; (*AO Blow-by Blower Percentage value to FC [%]*) (*OldName:new; Cycle:5*)
		rP_Red_Pr_CC_Norm : REAL; (*power reduction due to crank case pressure [% Pnom]*) (*OldName:ssPowerRed_Pr_CC; Cycle:5*)
		tBbBlower : HALioDo_Type; (*DO Blow-by Blower*) (*OldName:new; Cycle:5*)
		tECWP_Service : HALioDo_Type; (*DO engine cooling water service pump*) (*OldName:DI_ECWP_Service; Cycle:5*)
		rT_EO_PreH : REAL; (*engine oil temperature preheating*) (* Oldname: newPV, Cycle:5 *)
		STP_STRT : BOOL; (* tooth to tooth --> air starter off *) (*Oldname: newPV, Cycle:5*) (*V04.04.00.00*)
		tTCOP_GridOk : HALioDo_Type; (*TC oil pump power supply ok*) (*OldName:DI_TCOP_NETZ; Cycle:5;*)
		tManAuxCtr : tManAuxCtr_typ; (*Manual operating auxiliaries control - Handbedienebene*) (*OldName: new PV; Cycle: 5;*)
		bTC_CoolDownRun : BOOL; (*TC post cooling is demanded*) (*OldName: newPV; Cycle: 5;*)
		tGearPump_Dem : HALioDo_Type; (*gear pump demand*) (*OldName:A_GEKP; Cycle:5;*)
		tOFUP_Centrifuge : HALioDo_Type; (*oil filter unit pump centrifuge M.03-P-006*) (* Oldname:newPV;Cycle:5*)
		tOFUP_Filter : HALioDo_Type; (*oil filter unit pump filter M.03-P-007*) (* Oldname:newPV;Cycle:5*)
		bPreL_FS_EngStaRel : BOOL; (*prelubrication engine fast start release*) (* Oldname:newPV;Cycle:5*)
		bEOP_OilPumpFail : BOOL; (*Oil pump defective, oil pump monitoring *) (* Oldname:newPV;Cycle:5*)
		tTCOV_CoClose : HALioDo_Type; (*TC oil valve command close*) (*OldName:newPV; Cycle:5;*)
		bPreL_FS_Act : BOOL; (*permanent prelubrication activ*) (*OldName:newPv; Cycle:5;*)
		bOilskidDemSTFS : BOOL; (*oilskid demand for slowturn faststart*) (* Oldname: new PV, Cycle:5 *)
		bACP_AirER_Dem : BOOL; (* Active Cooling Program Room Air Ventilation demanded *) (*OldName:newPv; Cycle:5;*)
		tACP_AirER_Dem : HALioDo_Type; (* Active Cooling Program Room Air Ventilation demanded *) (*OldName:newPv; Cycle:5;*)
		tACP_HT_Dem : HALioDo_Type; (*Active Cooling Program - High Temperature demanded*) (*OldName:newPv; Cycle:5;*)
		rCustomizedAG : ARRAY[0..99]OF REAL; (*New customizable interface 2017  - BETA PHASE, use only in coordination with TPSS*)
		iStartCount : UINT; (*Number of Start*)
		bT_EOP_RelFS : BOOL; (*Oil temperature release fast start*)
		tECW_HydrPreH_Pump_Dem : HALioDo_Type; (*DO Hydraulic ECW pre-heating pump demand*)
		tECW_HydrPreH_Val_DemOpen : HALioDo_Type; (*DO Hydraulic ECW pre-heating valve demand open*)
		tHWP1_Dem : HALioDo_Type; (*DO Redundant heating water pump 1 demand (P.06-M-001)*)
		tHWP2_Dem : HALioDo_Type; (*DO Redundant heating water pump 2 demand (P.06-M-002)*)
		tCCWP1_Dem : HALioDo_Type; (*DO Redundant charge cooler water pump 1 demand (P.07-M-003)*)
		tCCWP2_Dem : HALioDo_Type; (*DO Redundant charge cooler water pump 2 demand (P.07-M-013)*)
		tCC2WP1_Dem : HALioDo_Type; (*DO Redundant charge cooler 2 water pump 1 demand (P.07-M-007)*)
		tCC2WP2_Dem : HALioDo_Type; (*DO Redundant charge cooler 2 water pump 2 demand (P.07-M-017)*)
		tEmCWP1_Dem : HALioDo_Type; (*DO Redundant emergency cooler water pump 1 demand (P.09-M-001)*)
		tEmCWP2_Dem : HALioDo_Type; (*DO Redundant emergency cooler water pump 2 demand (P.09-M-002)*)
		rDPr_OFU_Filt : REAL; (* Oilfilter difference pressure (oil filter unit) [bar] *)
		tAirST_ValEngage : HALioDo_Type; (*DO Air starter valve engage (E.31-YCS-001)*)
		tAirST_ValStart : HALioDo_Type; (*DO Air starter valve start (E.31-YCS-002)*)
		bAMM_Pr_AirStarter_Tank_Lo : BOOL; (*Air starter compressed air tank pressure low (for DAI)*)
		tFreshOilPump_Block : HALioDo_Type; (*DO Oil pressure max. Block fresh oil pump*)
		bNoExtendedPrelube : BOOL; (*No extended prelubrication active (allows 5min start)*)
		tBufferBat1_Disconnect : HALioDo_Type; (*DO Disconnect buffer battery 1*)
		tBufferBat2_Disconnect : HALioDo_Type; (*DO Disconnect buffer battery 2*)
		tBufferBat1_ConnectLoad : HALioDo_Type; (*DO Connect load resistor buffer battery 1*)
		tBufferBat2_ConnectLoad : HALioDo_Type; (*DO Connect load resistor buffer battery 2*)
		tStarterBat_ConnectLoad : HALioDo_Type; (*DO Connect load resistor starter battery*)
		bECWP_MechDriven : BOOL; (* CUSTOM for new Pr_ECW plausibility check: Mechanically driven ECWP on type3 or type2 *)
		bECW_Gnl_PreH_Dem : BOOL; (* general engine cooling water preheating demand (electric or hydraulic) *)
		tCtrlBat_Disconnect : ARRAY[1..iNum_CtrlBatMon]OF HALioDo_Type; (*DO Disconnect control battery*)
		tCtrlBat_ConnectLoad : ARRAY[1..iNum_CtrlBatMon]OF HALioDo_Type; (*DO Connect load resistor control battery*)
		bCust_EO_Level_Hi : BOOL; (*Bus signal for customer: Oil level max signal - oil overfill protection*) (*OldName:newPv; Cycle:5;*) (*V04.13.00.00*)
		bSt_RelAuxOff_STT_op : BOOL; (*Starter temperature release off for op_state and CBM*)
		bInLouDemAG : BOOL; (*Inlet louver demand for purge cranking cycle for fast start*)
		bFS_Rdy_STT_StPurge : BOOL; (*purge state and starter temperature readiness for fast start*)
		iMissfCyl_PurgeCrk : UDINT; (*skip fire order for all cylinders while purging*)
		bMissfCyl_PurgeCrk : BOOL; (*skip fire all cylinders while purging*)
		bEleStarter_Dem_PurgeCrkCyl : BOOL; (*starter demand during purge cranking cycle*)
		bEleStarter_Dem_PurgeCrkCylFS : BOOL; (*starter demand during purge cranking cycle for FS preparation*)
	END_STRUCT;
	ParaOil_typ : 	STRUCT
		kwh : REAL;
		ucIndexOil : USINT;
		OilCounter : ARRAY[0..19]OF tOilCounter;
	END_STRUCT;
	rtctime_typ : 	STRUCT
		year : UINT;
		month : USINT;
		day : USINT;
		reserve : USINT;
		hour : USINT;
		minute : USINT;
		second : USINT;
		millisec : UINT;
		microsec : UINT;
	END_STRUCT;
	tOilCounter : 	STRUCT
		oil_volume : DINT;
		delta_kwh : DINT;
		day : UINT;
		month : UINT;
		year : UINT;
		hour : UINT;
		minute : UINT;
		averaging : BOOL;
		Bh : DINT;
		rOC_Consum : REAL; (*Oil consumption during the last measurement (volume / kwh)*)
		rP_OC_Avg : REAL; (*Average power during the last measurement*)
		rOC_DeltaOpHour : REAL; (*Operating hours during last measurement*)
	END_STRUCT;
	VIS2MM_struct : 	STRUCT
		bDem_Oil_Filling : BOOL; (*HMI Demand fresh oil pump start for oil filling*) (*OldName: NewPv V4.14*)
		bDem_StopOil_Filling : BOOL; (*HMI Stop Demand for oil pumpst for oil filling/exchange*) (*OldName: NewPv V4.14*)
		bDem_Oil_Change : BOOL; (*HMI Demand waste oil pump start for oil exchange*) (*OldName: NewPv V4.14*)
		bEO_Change_Dem : BOOL; (*HMI demand of oil filling pump (button) *) (*OldName:new in V4.14; Cycle:5*)
		tCtr_CC_In : _tGeACtrIn; (*actual speed BlowBy*) (*OldName:new; Cycle:5*)
		tCtr_ECW_In : _tGeACtrIn; (*engine cooling water controller*) (*OldName:new; Cycle:5*)
		bEOP_DemMan : BOOL; (*bEOP_DemMan*) (*OldName:new; Cycle:5*)
		bHornOff : BOOL; (*horn off (button) from VIS*) (*OldName:new; Cycle:5*)
		tCtr_EOVal_In : _tGeACtrIn; (*engine oil cooler valve controller*) (*OldName:new; Cycle:5*)
		tCtr_EOVal_LT_In : _tGeACtrIn; (*engine oil cooler LT valve controller*) (*OldName:new; Cycle:5*)
		tManAuxCtr : tManAuxCtr_typ; (*Manual operating auxiliaries control - Handbedienebene*) (*OldName: new PV; Cycle: 5;*)
		bACP_Active : BOOL; (* Active Cooling Program active *)
		bACP_ECW_Active : BOOL; (* Active Cooling Program Engine Engine Cooling Water active *)
		bACP_EO_Active : BOOL; (* Active Cooling Program Engine Oil active *)
		bACP_AirER_Active : BOOL; (* Active Cooling Program Room Air active *)
		iACP_Year : UINT; (* Active Cooling Program - Automatic activation DateTime - Year *)
		iACP_Month : UINT; (* Active Cooling Program - Automatic activation DateTime - Month *)
		iACP_Day : UINT; (* Active Cooling Program - Automatic activation DateTime - Day *)
		iACP_Hour : UINT; (* Active Cooling Program - Automatic activation DateTime - Hour *)
		iACP_Minute : UINT; (* Active Cooling Program - Automatic activation DateTime - Minute *)
		iCnt_TC_abs : DINT; (* absolute counter *)
		iCnt_TC_rel_A : DINT; (* relative counter for failed TC post-cooling at bank A *)
		iCnt_TC_rel_B : DINT; (* relative counter for failed TC post-cooling at bank B *)
		iCnt_TC_abs_RSP : DINT; (* absolute counter for failed TC post-cooling caused by a DIANE power supply interruption *)
		bOilExchange : BOOL; (*Oil exchanged (button) from VIS*)
		bOilSample : BOOL; (*Oil sample taken (button) from VIS*)
		iOilSampleOh : DINT; (*reset value for oil sample counter*)
		bCWExchange : BOOL; (*cooling water exchanged (button) from VIS*)
		bCWSample : BOOL; (*cooling water sample taken (button) from VIS*)
		iCWSampleOh : DINT; (*reset value for cooling water sample counter*)
		bBatMon_ManTestStart : BOOL; (*Manual request for start of buffer battery test*)
		bCtrlBatMon_ManTestStart : BOOL; (*Manual request for start of control battery test*)
		iOQS_OC_OilTypeIdx : UINT; (*Oil quality sensor: oil type selection*)
		bOQS_OC_ConfigOilType : BOOL; (*Oil quality sensor: change configuration of oil type*)
		bOQS_OC_ReadOilType : BOOL; (*Oil quality sensor: read configuration of oil type*)
		bOQS_OilSampleOh_Man : BOOL; (*Oil quality sensor: Activate manual oil sampling interval*)
	END_STRUCT;
	tManAuxCtr_typ : 	STRUCT
		bGnl_Rel : BOOL; (*General release. Safety conditions (gas alarm, fire alarm, safety loop, ..) are OK.*) (*OldName: new PV; Cycle: 5;*)
		bECWP_PreH_COf_Man : BOOL; (*engine cooling water pump preheating demand off*) (*OldName: new PV; Cycle: 5;*)
		bECW_PreH_COf_Man : BOOL; (*engine cooling water preheating demand off*) (*OldName: new PV; Cycle: 5;*)
		bInAirER_Lou2DemOpen_Man : BOOL; (*demand open air inlet louver 2*) (*OldName: new PV; Cycle:5;*)
		bInAirER_Lou1DemOpen_Man : BOOL; (*demand open air inlet louver 1*) (*OldName: new PV; Cycle:5;*)
		bOutAirER_LouDemOpen_Man : BOOL; (*open air outlet louver *) (*OldName: new PV; Cycle:5;*)
		bInAirER_Fan1DemOn_Man : BOOL; (*demand air inlet ventilator 1*) (*OldName: new PV; Cycle:5;*)
		bInAirER_Fan2DemOn_Man : BOOL; (*demand air inlet ventilator 2*) (*OldName: new PV; Cycle:5;*)
		bER_FC_Set_Man : BOOL; (*demand engine room frequency converter setpoint*) (*OldName: new PV; Cycle:5;*)
		rER_FC_Set_Man : REAL; (*engine room frequency converter setpoint [%]*) (*OldName: new PV; Cycle:5;*)
		bER_OutlV_FC_Set_Man : BOOL; (*demand engine room air outlet ventilation frequency converter setpoint*) (*OldName: new PV; Cycle:5;*)
		rER_OutlV_FC_Set_Man : REAL; (*engine room air outlet ventilation frequency converter setpoint [%]*) (*OldName: new PV; Cycle:5;*)
		bEC_DemPump_Man : BOOL; (*emergency cooler demand pump*) (*OldName: new PV; Cycle:5;*)
		bEC_DemFan_Man : BOOL; (*emergency cooler demand fan 1 - 16*) (*OldName: new PV; Cycle:5;*)
		bChC_DemPump_Man : BOOL; (*charge cooler demand pump*) (*OldName: new PV; Cycle:5;*)
		bChC_DemFan_Man : BOOL; (*charge cooler demand fan 1 - 16*) (*OldName: new PV; Cycle:5;*)
		bEG_BoVaCoOpen_Man : BOOL; (*exhaust gas boiler valve command open*) (*OldName: new PV; Cycle:5;*)
		bEG_BoVaCoClose_Man : BOOL; (*exhaust gas boiler valve command close*) (*OldName: new PV; Cycle:5;*)
		bEG_ByVaCoOpen_Man : BOOL; (*exhaust gas bypass valve command open*) (*OldName: new PV; Cycle:5;*)
		bEG_ByVaCoClose_Man : BOOL; (*exhaust gas bypass valve command close*) (*OldName: new PV; Cycle:5;*)
		bAuxCust_Man : ARRAY[0..40]OF BOOL; (*reserve customer auxiliaries*) (*OldName: new PV; Cycle:5;*)
		bCDP_Dem_Man : BOOL; (*demand condensor pump*) (*OldName: new PV; Cycle:5;*)
		bBHV_Dem_Man : BOOL; (*demand boiler house ventilation*) (*OldName: newPv; Cycle:5;*)
		bHWF_Dem_Man : BOOL; (*demand heating circuit flap*) (*OldName:newPv; Cycle:5;*)
		bChC_Heating_Man : BOOL; (*charge cooler pre heating*) (*OldName:newPv; Cycle:5;*)
		bCO2_DemCodinox_Man : BOOL; (*CO2 demand CODINOX*) (*OldName:newPv; Cycle:5;*)
		bECWP_PreH_COf : BOOL; (*engine cooling water pump preheating demand off*) (*OldName: new PV; Cycle: 5;*)
		bECW_PreH_COf : BOOL; (*engine cooling water preheating demand off*) (*OldName: new PV; Cycle: 5;*)
		bInAirER_Lou2DemOpen : BOOL; (*demand open air inlet louver 2*) (*OldName: new PV; Cycle:5;*)
		bInAirER_Lou1DemOpen : BOOL; (*demand open air inlet louver 1*) (*OldName: new PV; Cycle:5;*)
		bOutAirER_LouDemOpen : BOOL; (*open air outlet louver *) (*OldName: new PV; Cycle:5;*)
		bInAirER_Fan1DemOn : BOOL; (*demand air inlet ventilator 1*) (*OldName: new PV; Cycle:5;*)
		bInAirER_Fan2DemOn : BOOL; (*demand air inlet ventilator 2*) (*OldName: new PV; Cycle:5;*)
		bER_OutlV_FC_Set : BOOL; (*demand engine room air outlet ventilation frequency converter setpoint*) (*OldName: new PV; Cycle:5;*)
		rER_OutlV_FC_Set : REAL; (*engine room air outlet ventilation frequency converter setpoint [%]*) (*OldName: new PV; Cycle:5;*)
		bER_FC_Set : BOOL; (*demand engine room frequency converter setpoint*) (*OldName: new PV; Cycle:5;*)
		rER_FC_Set : REAL; (*engine room frequency converter setpoint [%]*) (*OldName: new PV; Cycle:5;*)
		bEC_DemPump : BOOL; (*emergency cooler demand pump*) (*OldName: new PV; Cycle:5;*)
		bEC_DemFan : BOOL; (*emergency cooler demand fan 1 - 16*) (*OldName: new PV; Cycle:5;*)
		bChC_DemPump : BOOL; (*charge cooler demand pump*) (*OldName: new PV; Cycle:5;*)
		bChC_DemFan : BOOL; (*charge cooler demand fan 1 - 16*) (*OldName: new PV; Cycle:5;*)
		bEG_BoVaCoOpen : BOOL; (*exhaust gas boiler valve command open*) (*OldName: new PV; Cycle:5;*)
		bEG_BoVaCoClose : BOOL; (*exhaust gas boiler valve command close*) (*OldName: new PV; Cycle:5;*)
		bEG_ByVaCoOpen : BOOL; (*exhaust gas bypass valve command open*) (*OldName: new PV; Cycle:5;*)
		bEG_ByVaCoClose : BOOL; (*exhaust gas bypass valve command close*) (*OldName: new PV; Cycle:5;*)
		bAuxCust : ARRAY[0..70]OF BOOL; (*reserve customer auxiliaries*) (*OldName: new PV; Cycle:5;*)
		bCDP_Dem : BOOL; (*demand condensor pump*) (*OldName: new PV; Cycle:5;*)
		bBHV_Dem : BOOL; (*demand boiler house ventilation*) (*OldName: newPv; Cycle:5;*)
		bHWF_Dem : BOOL; (*demand heating circuit flap*) (*OldName:newPv; Cycle:5;*)
		bChC_Heating : BOOL; (*charge cooler pre heating*) (*OldName:newPv; Cycle:5;*)
		bCO2_DemCodinox : BOOL; (*CO2 demand CODINOX*) (*OldName:newPv; Cycle:5;*)
		bChC2_DemPump : BOOL; (*charge cooler 2 demand pump*) (*OldName: new PV; Cycle:5;*)
		bChC2_DemPump_Man : BOOL; (*charge cooler 2 demand pump*) (*OldName: new PV; Cycle:5;*)
		bChC2_DemFan : BOOL; (*charge cooler 2 demand fan 1 - 16*) (*OldName: new PV; Cycle:5;*)
		bChC2_DemFan_Man : BOOL; (*charge cooler 2 demand fan 1 - 16*) (*OldName: new PV; Cycle:5;*)
		bChC2_Heating : BOOL; (*charge cooler 2 pre heating*) (*OldName:newPv; Cycle:5;*)
		bChC2_Heating_Man : BOOL; (*charge cooler 2 pre heating*) (*OldName:newPv; Cycle:5;*)
		bECW_HydrPreH_COf : BOOL; (*engine cooling water hydraulic preheating demand off*) (*OldName: new PV; Cycle: 5;*)
		bECW_HydrPreH_COf_Man : BOOL; (*engine cooling water hydraulic preheating demand off*) (*OldName: new PV; Cycle: 5;*)
		bEOP_DemPump : BOOL; (*engine prelubrication pump manual demand*) (*OldName: new PV; Cycle: 5;*)
		bEOP_DemPump_Man : BOOL; (*engine prelubrication pump manual demand*) (*OldName: new PV; Cycle: 5;*)
	END_STRUCT;
	Perm_AG_Struct : 	STRUCT
		iCntH : DINT; (*service mode counter operating hours*)
		iCntS : DINT; (*service mode counter starts*)
		iCnt_TC_abs : DINT; (*absolute counter for failed post cooling of the turbocharger*)
		iCnt_TC_rel_A : DINT; (*relative counter for failed post cooling of the turbocharger on bank A*)
		iCnt_TC_rel_B : DINT; (*relative counter for failed post cooling of the turbocharger on bank B*)
		iCnt_TC_abs_RSP : DINT; (*absolute counter for failed post cooling of the turbocharger caused by DIANE power interruption*)
		iSt_TC_PwrInterrupt : DINT; (*permanent variable for TC black sut-down interruption by PLC power supply failure*)
		iOQS_OilSampleOh_Man : DINT; (*Oil quality sensor: Activate manual oil sampling interval*)
		iOQS_OC_OilTypeIdx : DINT; (*Oil quality sensor: oil type selection*)
		rTB_PermValue08 : REAL; (*spare permanent value for testbench- replace with new vars of same lenght, when needed*) (*OldName:new PV;Cycle:2;*)
		rTB_PermValue09 : REAL; (*spare permanent value for testbench- replace with new vars of same lenght, when needed*) (*OldName:new PV;Cycle:2;*)
		rTB_PermValue10 : REAL; (*spare permanent value for testbench- replace with new vars of same lenght, when needed*) (*OldName:new PV;Cycle:2;*)
		iOilSampleOh : DINT; (*reset value for oil sample counter*)
		iCnt_OilOh : DINT; (*Oil operating hours*)
		iCnt_OilSampleOh : DINT; (*Oil Operating hours until next sample*)
		tLastOilExchange : tFluidEvent; (*Last oil exchange information*)
		tLastOilSample : tFluidEvent; (*Last oil sample information*)
		iCWSampleOh : DINT; (*reset value for cooling water sample counter*)
		iCnt_CWOh : DINT; (*Cooling water operating hours*)
		iCnt_CWSampleOh : DINT; (*Cooling water operating hours until next sample*)
		tLastCWExchange : tFluidEvent; (*Last cooling water exchange information*)
		tLastCWSample : tFluidEvent; (*Last cooling water sample information*)
		bStartScavBgnFroce : BOOL; (*scavenging forced at the beginning of start attempt*)
		bStartScavFail : BOOL; (*Scavenging by starter motor failure*)
		bStartScavBgn : BOOL; (*Scavenging procedure anticipated at the beginning of the start attempt*)
		bSt_Purge : BOOL; (*Purge state (true: engine purged, false: engine not purged)*)
	END_STRUCT;
	tFluidEvent : 	STRUCT
		Oh_engine : DINT; (*Engine operting hours at fluid event [Oh]*)
		Oh_fluid : DINT; (*Fluid operating hours at fluid event [Oh]*)
		day : UINT; (*Day at fluid event*)
		month : UINT; (*Month at fluid event*)
		year : UINT; (*Year at fluid event*)
	END_STRUCT;
	tOQS_OC_OilConfig : 	STRUCT
		sData_OilCfgActive : STRING[iOQS_OC_OilSerialNr_CharSize]; (*oil type serial number string read from sensor*)
		sData_OilCfgUpd : STRING[iOQS_OC_OilCfg_CharSize]; (*oil type configuration string for writing to sensor*)
	END_STRUCT;
END_TYPE
```
